// SIMATIC STEP 7 (V5.x) project Formation_tolerie
// CPU: CPU
// station: Matériel
// station: API
// station: P_ADR_BUS
// station: P_ADR_BUS
// station: Configuration
// station: MOP
// program: Programme S7(1)
// program: Programme S7(2)

SYMBOL_TABLE
"I01"	DB 1	FB 1	// FACILITY: INSTANCE DB (FB1)
"I02"	DB 2	FB 2	// FACILITY: INSTANCE DB FOR MMC CONTROL (FB2)
"I03"	DB 3	FB 3	// FACILITY: INSTANCE DB FOR MOP/LOP
"I04"	DB 4	FB 4	// FACILITY: INSTANCE DB FOR COMMUNICATION / DB D'INSTANCE POUR LA COMMUNICATION
"SFM_DB"	DB 75	FB 20	// Bloc de diagnostic pour signalisation d'erreurs système
"SFM_GLOBAL_DB"	DB 76	DB 76	// Bloc de diagnostic pour signalisation d'erreurs système
"SFM_PN"	DB 77	DB 77	// PROFINET DIAGNOSTIC FUNCTION EDITING DB FOR IHMP
"IDENT"	DB 93	DB 93	// RFID DATAS / IDENTIFIANT DYNAMIQUE
"IIT"	DB 96	DB 96	// FACILITY: PART TABLE / DB TABLE PIECE
"IIS"	DB 97	DB 97	// FACILITY: SUPPORT WORD TABLE / DB MOTS SUPPORT
"IG"	DB 99	DB 99	// FACILITY: GLOBAL DB / DB GLOBAL
"Z1"	DB 100	FB 100	// ZONE 1: INSTANCE DB
"Z1A0"	DB 101	FB 101	// A0 ROBOT INSTANCE DATA BLOC / BLOC DE DONNEES INSTANCE A0 ROBOT
"Z1A01"	DB 102	FB 102	// A01 PREHENSEUR INSTANCE DATA BLOC / BLOC DE DONNEES INSTANCE A01 PREHENSEUR
"Z1B0"	DB 103	FB 103	// B0 MONTAGE INSTANCE DATA BLOC / BLOC DE DONNEES INSTANCE B0 MONTAGE
"Z1C0C"	DB 104	FB 104	// C0C CHGT_MEUBLE INSTANCE DATA BLOC / BLOC DE DONNEES INSTANCE C0C CHGT_MEUBLE
"Z1H0D"	DB 105	FB 105	// H0D DCHGT_MEUBL INSTANCE DATA BLOC / BLOC DE DONNEES INSTANCE H0D DCHGT_MEUBL
"Z1T"	DB 198	DB 198	// ZONE 1: REFERENCE TIME FOR MOVEMENTS
"Z1G"	DB 199	DB 199	// ZONE 1: GLOBAL DB
"ITS0"	DB 1100	FB 1100	// ILOT : DB INSTANCE FB1100
"ITSZ1_AU_ES_FZ"	DB 1110	FB 1110	// Z1 : DB D'INSTANCE DU FB 1110
"ITSZ1VAR"	DB 1113	FB 1113	// Z1 : DB D'INSTANCE DU FB 1113
"TSM"	DB 1279	DB 1279	// STD - DB global pour la Tâche de Sécurité
"TSE_AMONT"	DB 1286	FB 1692	// STD - INSTANCE DB OF FB 1692 (F_SENDDP) SAFETY DATA SEND
"TSR_AMONT"	DB 1287	FB 1693	// STD - INSTANCE DB OF FB 1693 (F_RCVDP) SAFETY DATA RECEIVE
"TSE_AVAL"	DB 1288	FB 1692	// STD - INSTANCE DB OF FB 1692 (F_SENDDP) SAFETY DATA SEND
"TSR_AVAL"	DB 1289	FB 1693	// STD - INSTANCE DB OF FB 1693 (F_RCVDP) SAFETY DATA RECEIVE
"F_GLOBDB"	DB 1300	DB 1300
"F00471__Z1RB1_M05"	DB 1301	FB 1300
"F00477__Z1RB1_M06"	DB 1302	FB 1300
"F00203__Z1ZB_M07"	DB 1303	FB 1300
"F00209__Z1ZB_M08"	DB 1304	FB 1300
"F00215__Z1ZB_M09"	DB 1305	FB 1300
"F00303__Z1SPA1"	DB 1306	FB 1300
"AFF"	DB 1863	DB 1863	// SIEBERT DISPLAY STRING STORAGE / STOCKAGE MESSAGE AFFICHEUR SIEBERT
"DB_IHM_WINCC"	DB 1962	FB 1962	// FACILITY: HMI INTERFACING WINCCFLEXIBLE RT
"DB_MMC"	DB 2000	DB 2000	// BACKUP COPY AND RESTORE OF EXTERN MEMORY MAP (MMC)
"DB_PN"	DB 2036	FB 2036	// INSTANCE IO PROFINET DB
"0_01_ILOT"	FB 1	FB 1	// FACILITY: FACILITY MANAGEMENT
"0_02_MMC"	FB 2	FB 2	// FACILITY: BACKUP MANAGEMENT AND DATA RESTITUTION ON EXTERNAL MMC CARD
"0_03_XOP"	FB 3	FB 3	// FACILITY: MOP/LOP MANAGEMENT
"0_04_COM"	FB 4	FB 4	// FACILITY: COM CONTROL WITH SIPTOL / GESTION DE LA COMMUNICATION AVEC SIPTOL
"SFM_FB"	FB 20	FB 20	// Bloc de diagnostic pour signalisation d'erreurs système
"1_00_ZONE1"	FB 100	FB 100	// ZONE 1: ZONE CONTROL
"1_A0_ROBOT"	FB 101	FB 101	// A0 ROBOT FUNCTION BLOC / SECTION PROGRAMME A0 ROBOT
"1_A01_PREHENSEUR"	FB 102	FB 102	// A01 PREHENSEUR FUNCTION BLOC / SECTION PROGRAMME A01 PREHENSEUR
"1_B0_MONTAGE"	FB 103	FB 103	// B0 MONTAGE FUNCTION BLOC / SECTION PROGRAMME B0 MONTAGE
"1_C0C_CHGT_MEUBLE"	FB 104	FB 104	// C0C CHGT_MEUBLE FUNCTION BLOC / SECTION PROGRAMME C0C CHGT_MEUBLE
"1_H0D_DCHGT_MEUBL"	FB 105	FB 105	// H0D DCHGT_MEUBL FUNCTION BLOC / SECTION PROGRAMME H0D DCHGT_MEUBL
"F_TON"	FB 185	FB 185	// F_: Timer Switch On Delay
"F_TOF"	FB 186	FB 186	// F_: Timer Switch Off Delay
"TS0"	FB 1100	FB 1100	// ILOT: FB Gestion SAFETY ilot
"TSZ1_AU_ES_FZ"	FB 1110	FB 1110
"F_IO_CGP"	FB 1300	FB 1300
"F_CTRL_1"	FB 1301	FB 1301
"F_CTRL_2"	FB 1302	FB 1302
"FITON"	FB 1303	FB 1303
"FIACK_GL"	FB 1304	FB 1304
"F_DIAG_N"	FB 1306	FB 1306
"F_RTGCO2"	FB 1308	FB 1308
"BF_DEVERM"	FB 1649	FB 1649	// BF STAGE DRY RUN CONTROL / BF GESTION DEVERMINAGE POSTE
"BF_RB_NISSAN"	FB 1650	FB 1650	// FANUC NISSAN ROBOT FB / BF ROBOT FANUC NISSAN
"TUSEND"	FB 1681	FB 1681	// Send Data via UDP
"TCON"	FB 1685	FB 1685	// Connect
"F_SENDDP"	FB 1692	FB 1692	// F_: Send Data via PROFIBUS DP / PROFINET IO
"F_RCVDP"	FB 1693	FB 1693	// F_: Receive Data via PROFIBUS DP / PROFINET IO
"F_ACK_GL"	FB 1695	FB 1695	// Acquittement global de toutes les périphéries F d'un groupe d'exécution F
"P_SEND"	FB 1698	FB 1698	// Send Data to CP340
"P_RCV"	FB 1699	FB 1699	// Receive Data from CP340
"BFS_BSEC1"	FB 1710	FB 1710
"BFS_BSECTR1"	FB 1711	FB 1711
"BFS_PORTE1"	FB 1712	FB 1712
"BFS_AIR1"	FB 1713	FB 1713
"BFS_CRM1"	FB 1714	FB 1714
"BFS_CR1"	FB 1715	FB 1715
"BFS_CAME_ROBOT1"	FB 1716	FB 1716
"BFS_MUT1"	FB 1717	FB 1717
"BFS_BIMA"	FB 1719	FB 1719
"BFS_ROB_KUKA_PS"	FB 1720	FB 1720
"BF_PNPN_MESG"	FB 1852	FB 1852	// SEND RECEIVE MESSAGE BY PNPN INTERFACE/ EMISSION RECEPTION MESSAGE VIA PNPN
"BF_G120DS_V2"	FB 1853	FB 1853	// G120D DRIVE BOX CONTROL / GESTION COFFRET VAR G120D
"BF_G120S_V2"	FB 1854	FB 1854	// G120 DRIVE PLATE CONTROL / GESTION PLATINE VAR G120
"BF_CARACT_SIEBERT"	FB 1856	FB 1856	// SIEBERT DISPLAY MESSAGE CONFIGURATION / MISE EN FORME MESSAGE AFFICHEUR SIEBERT
"BF_AFF SIEBERT (2*13) PN"	FB 1860	FB 1860	// AFFICHEUR 2 LIGNES DE 13 CARACTERES
"BF_WELDING_BOX"	FB 1868	FB 1868	// WELDING BOX CONTROL / GESTION DES COFFRETS PARAMETRES SOUDURE
"BF_CONF_MACHINE"	FB 1869	FB 1869	// GESTION BASE DE DONNEE CONFIGURATION MACHINE
"BF_CODE_PROCESS"	FB 1870	FB 1870	// GESTION BASE DE DONNEE CODE PROCESS
"BF_DATABASE3"	FB 1871	FB 1871	// DATABASE MANAGEMENT / GESTION BASE DE DONNEES
"BF_IHMMUT1"	FB 1874	FB 1874	// Diagnostic IHM(P) BFS_MUT1
"BF_IHMCAME_ROBOT1"	FB 1875	FB 1875	// BF gérant le bon fonctionnement de la came robot
"BF_IHMCR1"	FB 1876	FB 1876	// BF gérant l'IHM du relais non piloté par l'API mais controlé
"BF_IHMCRM1"	FB 1877	FB 1877	// BF gérant l'IHM du relais de controçle raccordement de masse CRM
"BF_CABRS"	FB 1897	FB 1897	// BARCODE READER / LECTEUR DE CODE A BARRE
"BF_IHMPORTE1"	FB 1930	FB 1930	// BF - ZONE : Diagnostic du bloc BFS_IHMPORTE
"BF_IHMAIR1"	FB 1931	FB 1931	// BF - ZONE : Diagnostic du bloc BFS_IHMAIR
"BF_ZONE_MODE_IHM1"	FB 1932	FB 1932	// Zone: Traitement des Modes et des pupitre de cde manu de la  zone
"BF_RB_COD_PREH_API"	FB 1953	FB 1953	// Gestion du préhenseur par API (séquences 1 à 16)
"BF_MODBUS_MASTER_CP340"	FB 1958	FB 1958	// MODBUS MAITRE SUR CP 340 (LIAISON SERIE)
"BF_MODBUS_SLAVE_CP340"	FB 1959	FB 1959	// MODBUS ESCLAVE AVEC CP340
"BF_MODBUS_TCPIP_MASTER"	FB 1960	FB 1960	// BF gerant le protocole MODBUS TCP/IP en tant que Client TCP et Maitre MODBUS
"BF_MODBUS_TCPIP_SLAVE"	FB 1961	FB 1961	// ESCLAVE MODBUS SUR CP ETHERNET
"BF_IHM_WINCC"	FB 1962	FB 1962	// BF- GESTION IMAGES WINCC FLEXIBLE
"BF_RB_SERVICE"	FB 1997	FB 1997	// BF- Envoi d'un groupe de robot en rodage
"BF_MMC"	FB 2000	FB 2000	// SAUVEGARDE ET RESTITUTION MEMOIRE SUR CARTE MEMOIRE EXTERNE (MMC)
"BF_MB_CHAINE1"	FB 2001	FB 2001	// PILOTAGE DU MOTEUR DU MEUBLE ET SURVEILLANCE DES DEFAUTS
"BF_MB_BUTEE1"	FB 2002	FB 2002	// MEUBLE A ACCUMULATION - PILOTAGE D'UNE BUTEE
"BF_ILOT"	FB 2004	FB 2004	// BF- GESTION INFO LIE A L'INSTALLATION (ILOT)
"BF_B_VIEAPI"	FB 2006	FB 2006	// CONTRÔLE DE LA COMMUNICATION ENTRE DEUX AUTOMATES EN LIAISON
"BF_BUTEE_CONVOYEUR2"	FB 2007	FB 2007	// PILOTAGE D'UNE BUTEE
"BF_IDENT"	FB 2015	FB 2015	// LECTURE/ECRITURE DES ETIQUETTES RFID
"BF_ROBOT"	FB 2016	FB 2016	// Interface API - Robot Version 1.2a
"BF_TCY_SUIV"	FB 2019	FB 2019	// MESURE LES TEMPS DE CYCLE D'UN MOYEN DE PRODUCTION
"BF_RUP_FLU"	FB 2020	FB 2020	// SUIVI-RUPTURE DE FLUX
"BF_CPT_PIECE"	FB 2021	FB 2021	// BF- COMPTEUR DE PIECE
"BF_ACT_DESACT"	FB 2033	FB 2033	// BF- ACTIVATION DESACTIVATION D'UN IO DEVICE
"BF_DIAG_PROFINET"	FB 2036	FB 2036	// BF- DIAGNOSTIC PROFINET IO
"BF_TF_TP"	FB 2037	FB 2037	// TRANSFERT DE TABLE DE MEMOIRES PIECES
"BF_FIFO"	FB 2039	FB 2039	// ASSURE LA GESTION D'UNE PILE FIFO
"BF_MVSE2P1"	FB 2040	FB 2040	// GESTION D'UN MOUVEMENT SIMPLE EFFET 2 POSITIONS
"BF_MOUVMP1"	FB 2041	FB 2041	// GESTION D'UN MOUVEMENT MULTI POSITION
"BF_MOUV2P1"	FB 2042	FB 2042	// BF- GESTION D'UN MOUVEMENT A 2 POSITIONS
"0_00_CYCLE_ILOT"	FC 1	FC 1	// FACILITY: CALL OF FACILITY FB
"SFM_FC"	FC 22	FC 22	// Bloc de diagnostic pour signalisation d'erreurs système
"1_00_CYCLE_Z1"	FC 100	FC 100	// ZONE 1: CALL OF FB ZONE
"0_00_TSSAFETY"	FC 1100	FC 1100	// STD - FACILITY: EXECUTION F GROUP ASSOCIATE TO OB32 (NORMAL TASK)
"0_00_TSCYCLE"	FC 1101	FC 1101	// CALL OPERATOR NOT IN ZONE FB LINKED IN FACILITY
"C_CNTRL"	FC 1697	FC 1697	// Read Connection Diagnostic Information
"AG_SEND"	FC 1698	FC 1698	// AG SEND
"AG_RECV"	FC 1699	FC 1699	// AG RECEIVE
"BADI"	I 0.0	BOOL	// (MOP-IM.M01-02): BOUTON ANNULATION DEFAUT
"BRI"	I 0.1	BOOL	// (MOP-IM.M01-02): BOUTON REARMEMENT ILOT
"BMCY"	I 0.2	BOOL	// (MOP-IM.M01-02): BOUTON MARCHE CYCLE
"SMM"	I 0.3	BOOL	// (MOP-IM.M01-02): SELECTEUR MODE MANUEL
"SMA"	I 0.4	BOOL	// (MOP-IM.M01-02): SELECTEUR MODE AUTO
"Z1BMR1"	I 0.5	BOOL	// (MOP-IM.M01-02): BOUTON RECUL MOUVEMENT
"Z1BMA1"	I 0.6	BOOL	// (MOP-IM.M01-02): BOUTON AVANCE MOUVEMENT
"B0DAPL1"	I 78.0	BOOL	// (B0IM.B0E1): B0 DETECTEUR AVANCE PILOTE 1
"B0DAPL2"	I 78.1	BOOL	// (B0IM.B0E1): B0 DETECTEUR AVANCE PILOTE 2
"B0DFSR3"	I 78.2	BOOL	// (B0IM.B0E1): B0 DETECTEUR FERMETURE SERRAGE 3
"B0DFSR4"	I 78.3	BOOL	// (B0IM.B0E1): B0 DETECTION FERMETURE SERRAGE 4
"B0DRPL1"	I 78.4	BOOL	// (B0IM.B0E1): B0 DETECTEUR RECUL PILOTE 1
"B0DRPL2"	I 78.5	BOOL	// (B0IM.B0E1): B0 DETECTEUR RECUL PILOTE 2
"B0DOSR3"	I 78.6	BOOL	// (B0IM.B0E1): B0 DETECTEUR OUVERTURE SERRAGE 3
"B0DOSR4"	I 78.7	BOOL	// (B0IM.B0E1): B0 DETECTION OUVERTURE SERRAGE 4
"B0DPP"	I 79.0	BOOL	// (B0IM.B0E1): B0 DETECTEUR PRESENCE PIECE
"A01DFSR1"	I 80.0	BOOL	// (A01IM.E1): A01 DETECTEUR FERMETURE SERRAGE 1
"A01DFSR2"	I 80.1	BOOL	// (A01IM.E1): A01 DETECTEUR FERMETURE SERRAGE 2
"A01DFSR3"	I 80.2	BOOL	// (A01IM.E1): A01 DETECTEUR FERMETURE SERRAGE 3
"A01DOSR1"	I 80.4	BOOL	// (A01IM.E1): A01 DETECTEUR OUVERTURE SERRAGE 1
"A01DOSR2"	I 80.5	BOOL	// (A01IM.E1): A01 DETECTEUR OUVERTURE SERRAGE 2
"A01DOSR3"	I 80.6	BOOL	// (A01IM.E1): A01 DETECTEUR OUVERTURE SERRAGE 3
"A01DPP"	I 81.0	BOOL	// (A01IM.E1): A01 DETECTION PRESENCE PIECE
"Z1CCSC1"	I 200.0	BOOL	// (Z1ZB.M02): CONTROLE RETOUR COMMUN SECURITE AU (SC1)
"Z1CCES"	I 200.1	BOOL	// (Z1ZB.M02): CONTROLE RETOUR COMMUN SECURITE ES
"Z1CCFZ"	I 200.2	BOOL	// (Z1ZB.M02): CONTROLE RETOUR COMMUN SECURITE FZ
"Z1CCB24Z"	I 200.4	BOOL	// (Z1ZB.M02): RETOUR CONTROLE DISJONCTEUR 24V (24Z)
"Z1CCB24R"	I 200.5	BOOL	// (Z1ZB.M02): RETOUR CONTROLE DISJONCTEUR 24V (24R)
"Z1CCB24SC"	I 200.6	BOOL	// (Z1ZB.M02): RETOUR CONTROLE DISJONCTEUR 24V (SC)
"Z1CP7B"	I 201.0	BOOL	// (Z1ZB.M03): CONTROLE PRESSION 7 BARS
"Z1CRM"	I 201.1	BOOL	// (Z1ZB.M03): RETOUR RELAIS CONTROLE DE MASSE
"Z1BMCY"	I 202.0	BOOL	// (Z1ZB.M04): BOUTON MARCHE CYCLE
"BAUI"	I 203.0	BOOL	// (Z1ZB.M07): ARRET D'URGENCE ILOT
"Z1SSZ"	I 203.2	BOOL	// (Z1ZB.M07): SELECTEUR SECURITE ZONE
"Z1SPA1BMCY"	I 300.7	BOOL	// (Z1SPA1.I0): BOUTON MARCHE CYCLE
"Z1SPA1BDACY"	I 301.0	BOOL	// (Z1SPA1.I1): BOUTON DEMANDE ARRET CYCLE
"Z1SPA1SPES"	I 301.3	BOOL	// (Z1SPA1.I1): SELECTEUR EN SERVICE / HORS SERVICE PORTILLON
"Z1SPA1SS"	I 303.7	BOOL	// (Z1SPA1.SI0): SELECTEUR DE SECURITE
"Z1SPA1CFP"	I 304.0	BOOL	// (Z1SPA1.SI1): CONTROLE FERMETURE PORTE
"A0RC_READY"	I 350.0	BOOL	// (A0RB.E1): ROBOT PRET
"A0MOTORON"	I 350.1	BOOL	// (A0RB.E1): SOUS PUISSANCE
"A0AUTO"	I 350.2	BOOL	// (A0RB.E1): COMMUTATEUR EN AUTOMATIQUE
"A0MANU"	I 350.3	BOOL	// (A0RB.E1): COMMUTATEUR EN MANUEL
"A0REPLI"	I 350.4	BOOL	// (A0RB.E1): POSITION DE REPLI
"A0RAMVT"	I 350.7	BOOL	// (A0RB.E1): MOUVEMENT EN COURS
"A0HPR"	I 351.0	BOOL	// (A0RB.E1): HORS PRODUCTION
"A0AOP"	I 351.1	BOOL	// (A0RB.E1): APPEL OPERATEUR
"A0DE"	I 351.2	BOOL	// (A0RB.E1): DERIVE
"A0TC"	I 351.3	BOOL	// (A0RB.E1): TOP CYCLE
"A0AI"	I 351.4	BOOL	// (A0RB.E1): ARRET INDUIT
"A0APE"	I 351.5	BOOL	// (A0RB.E1): ARRET PROPRE EXPLOITATION
"A0APF"	I 351.6	BOOL	// (A0RB.E1): ARRET PROPRE FABRICATION
"A0APP"	I 351.7	BOOL	// (A0RB.E1): ARRET PROPRE PANNE
"A0OR1"	I 352.0	BOOL	// (A0RB.E2): ORDRE 1
"A0OR2"	I 352.1	BOOL	// (A0RB.E2): ORDRE 2
"A0OR3"	I 352.2	BOOL	// (A0RB.E2): ORDRE 3
"A0OR4"	I 352.3	BOOL	// (A0RB.E2): ORDRE 4
"A0OR5"	I 352.4	BOOL	// (A0RB.E2): ORDRE 5
"A0OR6"	I 352.5	BOOL	// (A0RB.E2): ORDRE 6
"A0OR7"	I 352.6	BOOL	// (A0RB.E2): ORDRE 7
"A0OR8"	I 352.7	BOOL	// (A0RB.E2): ORDRE 8
"A0OR9"	I 353.0	BOOL	// (A0RB.E2): ORDRE 9
"A0OR10"	I 353.1	BOOL	// (A0RB.E2): ORDRE 10
"A0OR11"	I 353.2	BOOL	// (A0RB.E2): ORDRE 11
"A0OR12"	I 353.3	BOOL	// (A0RB.E2): ORDRE 12
"A0OR13"	I 353.4	BOOL	// (A0RB.E2): ORDRE 13
"A0OR14"	I 353.5	BOOL	// (A0RB.E2): ORDRE 14
"A0OR15"	I 353.6	BOOL	// (A0RB.E2): ORDRE 15
"A0OR16"	I 353.7	BOOL	// (A0RB.E2): ORDRE 16
"A0CCHDE"	I 354.0	BOOL	// (A0RB.E3): INFO CHANGEUR DEVERROUILLE
"A0CCHVE"	I 354.1	BOOL	// (A0RB.E3): INFO CHANGEUR VERROUILLE
"A0CPO"	I 354.2	BOOL	// (A0RB.E3): DETECTEUR PRESENCE OUTIL
"A0CPADV"	I 354.3	BOOL	// (A0RB.E3): CONTROLE PRESSION D'AIR DE DEVERROUILLAGE
"A0CPAV"	I 354.4	BOOL	// (A0RB.E3): CONTROLE PRESSION D'AIR DE VERROUILLAGE
"A0CPAS"	I 354.5	BOOL	// (A0RB.E3): CONTROLE PRESSION D'AIR (EV DE SECURITE)
"A0COHSUP"	I 354.6	BOOL	// (A0RB.E3): CONTROLE OUTIL HORS SUPPORT
"A0CFRO_ES"	I 354.7	BOOL	// (A0RB.E3): CONTROLE FRO MISE EN SERVICE
"A0CFRO_ZF"	I 355.0	BOOL	// (A0RB.E3): CONTROLE FRO FERMETURE ZONE 1
"A0CPAIR"	I 355.1	BOOL	// (A0RB.E3): CONTROLE PRESSION AIR DU ROBOT
"A0P1KCP"	I 355.2	BOOL	// (A0RB.E3): KCP ROBOT - POIDS 1
"A0P2KCP"	I 355.3	BOOL	// (A0RB.E3): KCP ROBOT - POIDS 2
"A0P4KCP"	I 355.4	BOOL	// (A0RB.E3): KCP ROBOT - POIDS 4
"A0P8KCP"	I 355.5	BOOL	// (A0RB.E3): KCP ROBOT - POIDS 8
"A0P16KCP"	I 355.6	BOOL	// (A0RB.E3): KCP ROBOT - POIDS 16
"A0P32KCP"	I 355.7	BOOL	// (A0RB.E3): KCP ROBOT - POIDS 32
"A0ORO1"	I 358.0	BOOL	// (A0RB.E5): ORDRE OUTIL 1
"A0ORO2"	I 358.1	BOOL	// (A0RB.E5): ORDRE OUTIL 2
"A0ORO3"	I 358.2	BOOL	// (A0RB.E5): ORDRE OUTIL 3
"A0ORO4"	I 358.3	BOOL	// (A0RB.E5): ORDRE OUTIL 4
"A0ORO5"	I 358.4	BOOL	// (A0RB.E5): ORDRE OUTIL 5
"A0ORO6"	I 358.5	BOOL	// (A0RB.E5): ORDRE OUTIL 6
"A0ORO7"	I 358.6	BOOL	// (A0RB.E5): ORDRE OUTIL 7
"A0ORO8"	I 358.7	BOOL	// (A0RB.E5): ORDRE OUTIL 8
"A0ORO9"	I 359.0	BOOL	// (A0RB.E5): ORDRE OUTIL 9
"A0ORO10"	I 359.1	BOOL	// (A0RB.E5): ORDRE OUTIL 10
"A0ORO11"	I 359.2	BOOL	// (A0RB.E5): ORDRE OUTIL 11
"A0ORO12"	I 359.3	BOOL	// (A0RB.E5): ORDRE OUTIL 12
"A0ORO13"	I 359.4	BOOL	// (A0RB.E5): ORDRE OUTIL 13
"A0ORO14"	I 359.5	BOOL	// (A0RB.E5): ORDRE OUTIL 14
"A0ORO15"	I 359.6	BOOL	// (A0RB.E5): ORDRE OUTIL 15
"A0ORO16"	I 359.7	BOOL	// (A0RB.E5): ORDRE OUTIL 16
"A0OR17"	I 364.0	BOOL	// (A0RB.E8): ORDRE 17
"A0OR18"	I 364.1	BOOL	// (A0RB.E8): ORDRE 18
"A0OR19"	I 364.2	BOOL	// (A0RB.E8): ORDRE 19
"A0OR20"	I 364.3	BOOL	// (A0RB.E8): ORDRE 20
"A0OR21"	I 364.4	BOOL	// (A0RB.E8): ORDRE 21
"A0OR22"	I 364.5	BOOL	// (A0RB.E8): ORDRE 22
"A0OR23"	I 364.6	BOOL	// (A0RB.E8): ORDRE 23
"A0OR24"	I 364.7	BOOL	// (A0RB.E8): ORDRE 24
"A0OR25"	I 365.0	BOOL	// (A0RB.E8): ORDRE 25
"A0OR26"	I 365.1	BOOL	// (A0RB.E8): ORDRE 26
"A0OR27"	I 365.2	BOOL	// (A0RB.E8): ORDRE 27
"A0OR28"	I 365.3	BOOL	// (A0RB.E8): ORDRE 28
"A0OR29"	I 365.4	BOOL	// (A0RB.E8): ORDRE 29
"A0OR30"	I 365.5	BOOL	// (A0RB.E8): ORDRE 30
"A0OR31"	I 365.6	BOOL	// (A0RB.E8): ORDRE 31
"A0OR32"	I 365.7	BOOL	// (A0RB.E8): ORDRE 32
"C0CDOB1"	I 430.0	BOOL	// (C0CIM.E1): DETECTEUR OUVERTURE BUTEE 1
"C0CDSPB1"	I 430.1	BOOL	// (C0CIM.E1): DETECTEUR SUPPORT PRESENT BUTEE 1
"C0CDOB2"	I 430.2	BOOL	// (C0CIM.E1): DETECTEUR OUVERTURE BUTEE 2
"C0CDSPB2"	I 430.3	BOOL	// (C0CIM.E1): DETECTEUR SUPPORT PRESENT BUTEE 2
"C0CDFB1"	I 430.4	BOOL	// (C0CIM.E1): DETECTEUR FERMETURE BUTEE 1
"C0CDSMAX"	I 430.5	BOOL	// (C0CIM.E1): DETECTEUR SEUIL MAX
"C0CDFB2"	I 430.6	BOOL	// (C0CIM.E1): DETECTEUR FERMETURE BUTEE 2
"C0CDDZB2"	I 430.7	BOOL	// (C0CIM.E1): DETECTEUR DEVERROUILLAGE DE ZONE BUTEE 2
"C0DPP1B2"	I 431.0	BOOL	// (C0CIM.E2): DETECTEUR PRESENCE PIECE TYPE 1
"C0CSSC"	I 431.2	BOOL	// (C0CIM.E2): C0C SELECTEUR DE SECURITE
"C0DPP2B2"	I 431.4	BOOL	// (C0CIM.E2): DETECTEUR PRESENCE PIECE TYPE 2
"H0DSSD"	I 450.0	BOOL	// (H0DIM.I1): SELECTEUR DE SECURITE
"H0DDM1_OK"	I 451.0	BOOL	// (H0DIM.DME1): DEPART MOTEUR PRET
"H0DDM1_CDM"	I 451.1	BOOL	// (H0DIM.DME1): DEPART MOTEUR EN MARCHE
"H0DDM1_DF"	I 451.2	BOOL	// (H0DIM.DME1): DEPART MOTEUR EN DEFAUT
"H0DDM1_AL"	I 451.3	BOOL	// (H0DIM.DME1): DEPART MOTEUR EN ALARME
"H0DDOB8"	I 453.0	BOOL	// (H0DIM.E1): DETECTEUR OUVERTURE BUTEE 8
"H0DDSPB8"	I 453.1	BOOL	// (H0DIM.E1): DETECTEUR SUPPORT PRESENT BUTEE 8
"H0DDOB9"	I 453.2	BOOL	// (H0DIM.E1): DETECTEUR OUVERTURE BUTEE 9
"H0DDSPB9"	I 453.3	BOOL	// (H0DIM.E1): DETECTEUR SUPPORT PRESENT BUTEE 9
"H0DDFB8"	I 453.4	BOOL	// (H0DIM.E1): DETECTEUR FERMETURE BUTEE 8
"H0DDSIL"	I 453.5	BOOL	// (H0DIM.E1): DETECTEUR SILHOUETTE
"H0DDFB9"	I 453.6	BOOL	// (H0DIM.E1): DETECTEUR FERMETURE BUTEE 9
"H0DDDZB9"	I 453.7	BOOL	// (H0DIM.E1): DETECTEUR DEVERROUILLAGE DE ZONE BUTEE 9
"H0DPP1B9"	I 454.0	BOOL	// (H0DIM.E2): DETECTEUR PRESENCE PIECE TYPE 1
"H0DDSMIN"	I 454.2	BOOL	// (H0DIM.E2): DETECTEUR SEUIL MIN
"H0DSSP"	I 454.3	BOOL	// (H0DIM.E2): SELECTEUR DE SECURITE
"H0DPP2B9"	I 454.4	BOOL	// (H0DIM.E2): DETECTEUR PRESENCE PIECE TYPE 2
"H0DDSMAX"	I 454.6	BOOL	// (H0DIM.E2): DETECTEUR SEUIL MAX
"H0DLIMEF"	I 454.7	BOOL	// (H0DIM.E2): LIMITEUR D'EFFORT
"Z1RB1CCB24Z"	I 470.4	BOOL	// (Z1RB1.M02): RETOUR CONTROLE DISJONCTEUR 24V (24Z)
"Z1RB1CCB24R"	I 470.5	BOOL	// (Z1RB1.M02): RETOUR CONTROLE DISJONCTEUR 24V (24R)
"A0BAU"	I 471.0	BOOL	// (Z1RB1.M05): ARRET D'URGENCE ROBOT
"A0RBMS1"	IW 350	WORD	// WORD 1 GENERAL DATA / GENERALITES
"A0RBMS2"	IW 352	WORD	// WORD 2 ROBOT ORDERS / ORDRES ROBOT
"A0RBMS3"	IW 354	WORD	// WORD 3 GRIPPER AND TOOL CHANGER / PREHENSEUR ET CHANGEUR OUTIL
"A0RBMS4"	IW 356	WORD	// WORD 4 FAULT NUMBER / NUMERO DE DEFAUT
"A0RBMS5"	IW 358	WORD	// WORD 5 TOOL ORDERS/ ORDRES OUTIL
"A0RBMS6"	IW 360	WORD	// WORD 6
"A0RBMS7"	IW 362	WORD	// WORD 7
"A0RBMS8"	IW 364	WORD	// WORD 8
"BA0"	M 0.0	BOOL	// FACILITY: BIT ALWAYS OFF / ILOT: BIT TOUJOURS A 0
"BA1"	M 0.1	BOOL	// FACILITY: BIT ALWAYS ON / ILOT: BIT TOUJOURS A 1
"BA1LIEN"	M 0.2	BOOL	// FACILITY: BIT ALWAYS ON (LINK IN THE PROGRAMMING NETWORK)
"SHUNT"	M 0.3	BOOL	// BIT FOR BYPASS DURING FACILITY START UP / BIT SHUNT POUR LA MISE AU POINT
"PERSO"	M 0.4	BOOL	// NEED TO PERSONALIZE BY THE PROGRAMMER / EQUATION A PERSONNALISER
"POUB"	M 0.5	BOOL	// DUST BIN BIT / BIT POUBELLE
"SYSFROID"	M 0.7	BOOL	// DETECTING COLD START PLC (OB102) / DETECTION DEMARRAGE A FROID API (OB102)
"ICL080S"	M 1.4	BOOL	// BLINKING INFORMATION / INFORMATION CLIGNOTEMENT
"IADF"	M 10.1	BOOL	// FACILITY: FAULT RESET INFORMATION (SAFETY)
"IR"	M 10.2	BOOL	// FACILITY: CONTROL ON INFORMATION (SAFETY)
"Z1DEF_MAJ"	M 11.0	BOOL	// ZONE 1: MAJOR FAULT (SAFETY)
"Z1IADF"	M 11.1	BOOL	// ZONE 1: FAULT RESET INFORMATION (SAFETY)
"Z1IR"	M 11.2	BOOL	// ZONE 1: CONTROL ON INFORMATION (SAFETY)
"Z1IAFJ"	M 11.3	BOOL	// ZONE 1: END OF PRODUCTION STOP INFORMATION (SAFETY)
"Z1MAUTO"	M 11.4	BOOL	// ZONE 1: ZONE IN AUTOMATIC MODE (SAFETY)
"H0AV"	M 100.0	BOOL	// Pilotage chaine H0
"SIMU"	M 105.0	BOOL	// Mode simulation en cours
"CYCL_EXC"	OB 1	OB 1	// EXECUTION CYCLE
"CYC_INT4"	OB 34	OB 34	// CYCLIC INTERRUPT 4
"I/O_FLT1"	OB 82	OB 82	// I/O POINT FAULT 1
"I/O_FLT2"	OB 83	OB 83	// I/O POINT FAULT 2
"OBNL_FLT"	OB 85	OB 85	// OB NOT LOADED FAULT
"RACK_FLT"	OB 86	OB 86	// LOSS OF RACK FAULT
"COMPLETE RESTART"	OB 100	OB 100	// COMPLETE RESTART
"MOD_ERR"	OB 122	OB 122	// MODULE ACCESS ERROR
"VADI"	Q 0.0	BOOL	// (MOP-IM.M06-07): VOYANT ANNULATION DEFAUT
"VMCY"	Q 0.1	BOOL	// (MOP-IM.M06-07): VOYANT MARCHE CYCLE
"VAOP"	Q 0.3	BOOL	// (MOP-IM.M06-07): VERRINE APPEL OPERATEUR
"A01EFSR1"	Q 56.0	BOOL	// (A01IM.S1): EV FERMETURE SERRAGE 1
"A01EFSR2"	Q 56.1	BOOL	// (A01IM.S1): A01 EV FERMETURE SERRAGE 2
"A01EFSR3"	Q 56.2	BOOL	// (A01IM.S1): A01 EV FERMETURE SERRAGE 3
"A01EOSR1"	Q 56.4	BOOL	// (A01IM.S1): A01 OUVERTURE SERRAGE 1
"A01EOSR2"	Q 56.5	BOOL	// (A01IM.S1): A01 EV OUVERTURE SERRAGE 2
"A01EOSR3"	Q 56.6	BOOL	// (A01IM.S1): A01 EV OUVERTURE SERRAGE 3
"B0EAPL1"	Q 58.0	BOOL	// (B0IM.B0S1): B0 EV AVANCE PILOTE 1
"B0EAPL2"	Q 58.1	BOOL	// (B0IM.B0S1): B0 EV AVANCE PILOTE 2
"B0EFSR3"	Q 58.2	BOOL	// (B0IM.B0S1): B0 EV FERMETURE SERRAGE 3
"B0EFSR4"	Q 58.3	BOOL	// (B0IM.B0S1): B0 EV FERMETURE SERRAGE 4
"B0ERPL1"	Q 58.4	BOOL	// (B0IM.B0S1): B0 EV RECUL PILOTE 1
"B0ERPL2"	Q 58.5	BOOL	// (B0IM.B0S1): B0 EV RECUL PILOTE 2
"B0EOSR3"	Q 58.6	BOOL	// (B0IM.B0S1): B0 EV OUVERTURE SERRAGE 3
"B0EOSR4"	Q 58.7	BOOL	// (B0IM.B0S1): B0 EV OUVERTURE SERRAGE 4
"Z1VMCY"	Q 200.0	BOOL	// (Z1ZB.M05): VOYANT MARCHE CYCLE
"Z1RCM"	Q 200.7	BOOL	// (Z1ZB.M05): RELAIS DE CONTROLE DE MASSE
"Z1RSC1"	Q 215.0	BOOL	// (Z1ZB.M09): RELAI COMMUN DE SECURITE SC1
"Z1RES"	Q 215.1	BOOL	// (Z1ZB.M09): RELAI COMMUN DE SECURITE ES
"Z1RFZ"	Q 215.2	BOOL	// (Z1ZB.M09): RELAI COMMUN DE SECURITE FZ
"Z1SPA1VMCY"	Q 300.7	BOOL	// (Z1SPA1.O0): VOYANT MARCHE CYCLE
"Z1SPA1VDACY"	Q 301.0	BOOL	// (Z1SPA1.O1): VOYANT DEMANDE ARRET CYCLE
"A0AEVRB"	Q 350.0	BOOL	// (A0RB.S1): AUTORISATION D'EVOLUTION
"A0DMSP"	Q 350.1	BOOL	// (A0RB.S1): DEMANDE DE MISE SOUS PUISSANCE
"A0STOP"	Q 350.2	BOOL	// (A0RB.S1): ARRET ROBOT
"A0DDCY"	Q 350.3	BOOL	// (A0RB.S1): DEPART CYCLE
"A0DEV"	Q 350.4	BOOL	// (A0RB.S1): DEVERMINAGE
"A0CVC_0"	Q 350.5	BOOL	// (A0RB.S1): CONTROLE VALIDATION CODE A 0
"A0CVC_1"	Q 350.6	BOOL	// (A0RB.S1): CONTROLE VALIDATION CODE A 1
"A0CPCO"	Q 350.7	BOOL	// (A0RB.S1): CONTOLE PARITE CODE
"A0C1"	Q 351.0	BOOL	// (A0RB.S1): CODE POIDS 1
"A0C2"	Q 351.1	BOOL	// (A0RB.S1): CODE POIDS 2
"A0C4"	Q 351.2	BOOL	// (A0RB.S1): CODE POIDS 4
"A0C8"	Q 351.3	BOOL	// (A0RB.S1): CODE POIDS 8
"A0C16"	Q 351.4	BOOL	// (A0RB.S1): CODE POIDS 16
"A0C32"	Q 351.5	BOOL	// (A0RB.S1): CODE POIDS 32
"A0C64"	Q 351.6	BOOL	// (A0RB.S1): CODE POIDS 64
"A0C128"	Q 351.7	BOOL	// (A0RB.S1): CODE POIDS 128
"A0EV1"	Q 352.0	BOOL	// (A0RB.S2): EVENEMENT 1
"A0EV2"	Q 352.1	BOOL	// (A0RB.S2): EVENEMENT 2
"A0EV3"	Q 352.2	BOOL	// (A0RB.S2): EVENEMENT 3
"A0EV4"	Q 352.3	BOOL	// (A0RB.S2): EVENEMENT 4
"A0EV5"	Q 352.4	BOOL	// (A0RB.S2): EVENEMENT 5
"A0EV6"	Q 352.5	BOOL	// (A0RB.S2): EVENEMENT 6
"A0EV7"	Q 352.6	BOOL	// (A0RB.S2): EVENEMENT 7
"A0EV8"	Q 352.7	BOOL	// (A0RB.S2): EVENEMENT 8
"A0EV9"	Q 353.0	BOOL	// (A0RB.S2): EVENEMENT 9
"A0EV10"	Q 353.1	BOOL	// (A0RB.S2): EVENEMENT 10
"A0EV11"	Q 353.2	BOOL	// (A0RB.S2): EVENEMENT 11
"A0EV12"	Q 353.3	BOOL	// (A0RB.S2): EVENEMENT 12
"A0EV13"	Q 353.4	BOOL	// (A0RB.S2): EVENEMENT 13
"A0EV14"	Q 353.5	BOOL	// (A0RB.S2): EVENEMENT 14
"A0EV15"	Q 353.6	BOOL	// (A0RB.S2): EVENEMENT 15
"A0EV16"	Q 353.7	BOOL	// (A0RB.S2): EVENEMENT 16
"A0ENPRO"	Q 354.0	BOOL	// (A0RB.S3): EN PRODUCTION
"A0RFZ"	Q 354.1	BOOL	// (A0RB.S3): ZONE FERMEE
"A0GS1"	Q 356.0	BOOL	// (A0RB.S4): GROUPE SEQUENCE POIDS 1
"A0GS2"	Q 356.1	BOOL	// (A0RB.S4): GROUPE SEQUENCE POIDS 2
"A0GS4"	Q 356.2	BOOL	// (A0RB.S4): GROUPE SEQUENCE POIDS 4
"A0GS8"	Q 356.3	BOOL	// (A0RB.S4): GROUPE SEQUENCE POIDS 8
"A0E1_SRE"	Q 356.4	BOOL	// (A0RB.S4): INFO DETECTION RECUL SEQUENCE 1
"A0E1_SAV"	Q 356.5	BOOL	// (A0RB.S4): INFO DETECTION AVANCE SEQUENCE 1
"A0E2_SRE"	Q 356.6	BOOL	// (A0RB.S4): INFO DETECTION RECUL SEQUENCE 2
"A0E2_SAV"	Q 356.7	BOOL	// (A0RB.S4): INFO DETECTION AVANCE SEQUENCE 2
"A0DECH"	Q 357.0	BOOL	// (A0RB.S4): COMMANDE DEVERROUILLAGE CHANGEUR
"A0EVO1"	Q 358.0	BOOL	// (A0RB.S5): EVENEMENT OUTIL 1
"A0EVO2"	Q 358.1	BOOL	// (A0RB.S5): EVENEMENT OUTIL 2
"A0EVO3"	Q 358.2	BOOL	// (A0RB.S5): EVENEMENT OUTIL 3
"A0EVO4"	Q 358.3	BOOL	// (A0RB.S5): EVENEMENT OUTIL 4
"A0EVO5"	Q 358.4	BOOL	// (A0RB.S5): EVENEMENT OUTIL 5
"A0EVO6"	Q 358.5	BOOL	// (A0RB.S5): EVENEMENT OUTIL 6
"A0EVO7"	Q 358.6	BOOL	// (A0RB.S5): EVENEMENT OUTIL 7
"A0EVO8"	Q 358.7	BOOL	// (A0RB.S5): EVENEMENT OUTIL 8
"A0EVO9"	Q 359.0	BOOL	// (A0RB.S5): EVENEMENT OUTIL 9
"A0EVO10"	Q 359.1	BOOL	// (A0RB.S5): EVENEMENT OUTIL 10
"A0EVO11"	Q 359.2	BOOL	// (A0RB.S5): EVENEMENT OUTIL 11
"A0EVO12"	Q 359.3	BOOL	// (A0RB.S5): EVENEMENT OUTIL 12
"A0EVO13"	Q 359.4	BOOL	// (A0RB.S5): EVENEMENT OUTIL 13
"A0EVO14"	Q 359.5	BOOL	// (A0RB.S5): EVENEMENT OUTIL 14
"A0EVO15"	Q 359.6	BOOL	// (A0RB.S5): EVENEMENT OUTIL 15
"A0EVO16"	Q 359.7	BOOL	// (A0RB.S5): EVENEMENT OUTIL 16
"A0EV17"	Q 364.0	BOOL	// (A0RB.S8): EVENEMENT 17
"A0EV18"	Q 364.1	BOOL	// (A0RB.S8): EVENEMENT 18
"A0EV19"	Q 364.2	BOOL	// (A0RB.S8): EVENEMENT 19
"A0EV20"	Q 364.3	BOOL	// (A0RB.S8): EVENEMENT 20
"A0EV21"	Q 364.4	BOOL	// (A0RB.S8): EVENEMENT 21
"A0EV22"	Q 364.5	BOOL	// (A0RB.S8): EVENEMENT 22
"A0EV23"	Q 364.6	BOOL	// (A0RB.S8): EVENEMENT 23
"A0EV24"	Q 364.7	BOOL	// (A0RB.S8): EVENEMENT 24
"A0EV25"	Q 365.0	BOOL	// (A0RB.S8): EVENEMENT 25
"A0EV26"	Q 365.1	BOOL	// (A0RB.S8): EVENEMENT 26
"A0EV27"	Q 365.2	BOOL	// (A0RB.S8): EVENEMENT 27
"A0EV28"	Q 365.3	BOOL	// (A0RB.S8): EVENEMENT 28
"A0EV29"	Q 365.4	BOOL	// (A0RB.S8): EVENEMENT 29
"A0EV30"	Q 365.5	BOOL	// (A0RB.S8): EVENEMENT 30
"A0EV31"	Q 365.6	BOOL	// (A0RB.S8): EVENEMENT 31
"A0EV32"	Q 365.7	BOOL	// (A0RB.S8): EVENEMENT 32
"C0CEOB1"	Q 430.0	BOOL	// (C0CIM.S1): ELECTROVANNE OUVERTURE BUTEE 1
"C0CEOB2"	Q 430.1	BOOL	// (C0CIM.S1): ELECTROVANNE OUVERTURE BUTEE 2
"C0CEFB1"	Q 430.4	BOOL	// (C0CIM.S1): ELECTROVANNE FERMETURE BUTEE 1
"C0CEFB2"	Q 430.5	BOOL	// (C0CIM.S1): ELECTROVANNE FERMETURE BUTEE 2
"H0DDM1_OAV"	Q 451.0	BOOL	// (H0DIM.DMS1): RELAI MARCHE AVANCE DEPART MOTEUR
"H0DDM1_ORE"	Q 451.1	BOOL	// (H0DIM.DMS1): RELAI MARCHE RECUL DEPART MOTEUR
"H0DDM1_FRE"	Q 451.2	BOOL	// (H0DIM.DMS1): COMMANDE FREIN DEPART MOTEUR
"H0DDM1_IR"	Q 451.3	BOOL	// (H0DIM.DMS1): INFORMATION REARMEMENT DEPART MOTEUR
"H0DEOB8"	Q 453.0	BOOL	// (H0DIM.S1): ELECTROVANNE OUVERTURE BUTEE 8
"H0DEOB9"	Q 453.1	BOOL	// (H0DIM.S1): ELECTROVANNE OUVERTURE BUTEE 9
"H0DEFB8"	Q 453.4	BOOL	// (H0DIM.S1): ELECTROVANNE FERMETURE BUTEE 8
"H0DEFB9"	Q 453.5	BOOL	// (H0DIM.S1): ELECTROVANNE FERMETURE BUTEE 9
"A0RBME1"	QW 350	WORD	// WORD 1 GENERAL DATA AND CYCLE CODE / CODE CYCLE ET GENERALITES
"A0RBME2"	QW 352	WORD	// WORD 2 ROBOT EVENTS / EVENEMENTS ROBOT
"A0RBME3"	QW 354	WORD	// WORD 3 GENERAL DATAS / GENERALITES
"A0RBME4"	QW 356	WORD	// WORD 4 GRIPPER AND TOOL CHANGER / PREHENSEUR ET CHANGEUR OUTIL
"A0RBME5"	QW 358	WORD	// WORD 5 TOOL EVENTS / EVENEMENTS OUTIL
"A0RBME6"	QW 360	WORD	// WORD 6
"A0RBME7"	QW 362	WORD	// WORD 7
"A0RBME8"	QW 364	WORD	// WORD 8
"TP"	SFB 3	SFB 3	// GENERATE A PULSE
"TON"	SFB 4	SFB 4	// GENERATE AN ON DELAY
"TOF"	SFB 5	SFB 5	// GENERATE AN OFF DELAY
"RDREC"	SFB 52	SFB 52	// READ A PROCESS DATA RECORD
"WRREC"	SFB 53	SFB 53	// WRITE A PROCESS DATA RECORD
"RALRM"	SFB 54	SFB 54	// Receive Alarm Data
"SET_CLK"	SFC 0	SFC 0	// SET SYSTEM CLOCK
"READ_CLK"	SFC 1	SFC 1	// READ SYSTEM CLOCK
"RD_SINFO"	SFC 6	SFC 6	// READ OB START INFORMATION
"D_ACT_DP"	SFC 12	SFC 12	// DEACTIVATING AND ACTIVATING DP SLAVES
"DPRD_DAT"	SFC 14	SFC 14	// READ CONSISTENT DATA OF A STANDARD DP SLAVE
"DPWR_DAT"	SFC 15	SFC 15	// WRITE CONSISTENT DATA TO A STANDARD DP SLAVE
"ALARM_SQ"	SFC 17	SFC 17	// Generate Block-Related Messages with Acknowledgment
"BLKMOV"	SFC 20	SFC 20	// COPY VARIABLES
"FILL"	SFC 21	SFC 21	// INITIALIZE A MEMORY AREA
"TEST_DB"	SFC 24	SFC 24	// TEST DATA BLOCK
"DIS_AIRT"	SFC 41	SFC 41	// DELAY THE HIGHER PRIORITY INTERRUPTS AND ASYNCHRONOUS ERRORS
"EN_AIRT"	SFC 42	SFC 42	// ENABLE HIGHER PRIORITY INTERRUPTS AND ASYNCHRONOUS ERRORS
"STP"	SFC 46	SFC 46	// CHANGE THE CPU TO STOP
"RDSYSST"	SFC 51	SFC 51	// READ A SYSTEM STATUS LIST OR PARTIAL LIST
"WR_REC"	SFC 58	SFC 58	// WRITE DATA RECORD
"RD_REC"	SFC 59	SFC 59	// READ A DATA RECORD
"TIME_TCK"	SFC 64	SFC 64	// READ THE SYSTEM TIME
"GEO_LOG"	SFC 70	SFC 70	// DETERMINE LOGICAL ADDRESS
"READ_DBL"	SFC 83	SFC 83	// READ DATA BLOCK OUT OF LOAD MEMORY
"WRIT_DBL"	SFC 84	SFC 84	// WRITE DATA BLOCK IN LOAD MEMORY
"DEL_SI"	SFC 106	SFC 106	// Deleting Dynamically Assigned System Instances
"ALARM_DQ"	SFC 107	SFC 107	// Creating Acknowledgeable Block-related Message
"ALARM_D"	SFC 108	SFC 108	// Creating Acknowledged Block-related Message
"LIEN_PUP"	UDT 1988	UDT 1988	// Gestion des Modes et des pupitres de cde manu de la  zone (BF_ZONE_MODE_IHM)
"LIEN_ILOT"	UDT 2004	UDT 2004	// INFO CONTROL LINKED TO THE FACILITY (BF_ILOT)
"MOT_FONC_MP"	UDT 2041	UDT 2041	// INFO CONTROL OF A MOVEMENT (BF_MOUVMP1)
"MOT_FONC"	UDT 2042	UDT 2042	// INFO D'UN MOUVEMENT (BF_MOUV2P1,BF_MVSE2P1, BF_RB_COD_PREH_API)
"VAT_SIMU"	VAT 1	
"Essais"	VAT 2	
END_SYMBOL_TABLE

SYMBOL_TABLE
"I01"	DB 1	FB 1	// FACILITY: INSTANCE DB (FB1)
"I02"	DB 2	FB 2	// FACILITY: INSTANCE DB FOR MMC CONTROL (FB2)
"I03"	DB 3	FB 3	// FACILITY: INSTANCE DB FOR MOP/LOP
"I04"	DB 4	FB 4	// FACILITY: INSTANCE DB FOR COMMUNICATION / DB D'INSTANCE POUR LA COMMUNICATION
"SFM_DB"	DB 75	FB 20	// FACILITY: DB FAILURE MESSAGE (SFM_FB) LINK WITH PROFINET CONTROL
"SFM_GLOBAL_DB"	DB 76	DB 76	// DIAGNOSTIC BLOCK FOR THE SIGNALISATION OF THE SYSTEM ERRORS
"SFM_PN"	DB 77	DB 77	// PROFINET DIAGNOSTIC FUNCTION EDITING DB FOR IHMP
"IDENT"	DB 93	DB 93	// RFID DATAS / IDENTIFIANT DYNAMIQUE
"IIT"	DB 96	DB 96	// FACILITY: PART TABLE / DB TABLE PIECE
"IIS"	DB 97	DB 97	// FACILITY: SUPPORT WORD TABLE / DB MOTS SUPPORT
"IG"	DB 99	DB 99	// FACILITY: GLOBAL DB / DB GLOBAL
"Z1"	DB 100	FB 100	// ZONE 1: INSTANCE DB
"Z1A0"	DB 101	FB 101	// A0 ROBOT INSTANCE DATA BLOC / BLOC DE DONNEES INSTANCE A0 ROBOT
"Z1A01"	DB 102	FB 102	// A01 PREHENSEUR INSTANCE DATA BLOC / BLOC DE DONNEES INSTANCE A01 PREHENSEUR
"Z1B0"	DB 103	FB 103	// B0 MONTAGE INSTANCE DATA BLOC / BLOC DE DONNEES INSTANCE B0 MONTAGE
"Z1C0C"	DB 104	FB 104	// C0C CHGT_MEUBLE INSTANCE DATA BLOC / BLOC DE DONNEES INSTANCE C0C CHGT_MEUBLE
"Z1H0D"	DB 105	FB 105	// H0D DCHGT_MEUBL INSTANCE DATA BLOC / BLOC DE DONNEES INSTANCE H0D DCHGT_MEUBL
"Z1T"	DB 198	DB 198	// ZONE 1: REFERENCE TIME FOR MOVEMENTS
"Z1G"	DB 199	DB 199	// ZONE 1: GLOBAL DB
"ITS0"	DB 1100	FB 1100	// ILOT : DB INSTANCE FB1100
"ITSZ1_AU_ES_FZ"	DB 1110	FB 1110	// Z1 : DB D'INSTANCE DU FB 1110
"ITSZ1VAR"	DB 1113	FB 1113	// Z1 : DB D'INSTANCE DU FB 1113
"TSM"	DB 1279	DB 1279	// STD - DB global pour la Tâche de Sécurité
"TSE_AMONT"	DB 1286	FB 1692	// STD - INSTANCE DB OF FB 1692 (F_SENDDP) SAFETY DATA SEND
"TSR_AMONT"	DB 1287	FB 1693	// STD - INSTANCE DB OF FB 1693 (F_RCVDP) SAFETY DATA RECEIVE
"TSE_AVAL"	DB 1288	FB 1692	// STD - INSTANCE DB OF FB 1692 (F_SENDDP) SAFETY DATA SEND
"TSR_AVAL"	DB 1289	FB 1693	// STD - INSTANCE DB OF FB 1693 (F_RCVDP) SAFETY DATA RECEIVE
"F_GLOBDB"	DB 1300	DB 1300
"F00471__Z1RB1_M05"	DB 1301	FB 1300
"F00477__Z1RB1_M06"	DB 1302	FB 1300
"F00203__Z1ZB_M07"	DB 1303	FB 1300
"F00209__Z1ZB_M08"	DB 1304	FB 1300
"F00215__Z1ZB_M09"	DB 1305	FB 1300
"F00303__Z1SPA1"	DB 1306	FB 1300
"AFF"	DB 1863	DB 1863	// SIEBERT DISPLAY STRING STORAGE / STOCKAGE MESSAGE AFFICHEUR SIEBERT
"DB_IHM_WINCC"	DB 1962	FB 1962	// FACILITY: HMI INTERFACING WINCCFLEXIBLE RT
"DB_MMC"	DB 2000	DB 2000	// BACKUP COPY AND RESTORE OF EXTERN MEMORY MAP (MMC)
"DB_PN"	DB 2036	FB 2036	// INSTANCE IO PROFINET DB
"0_01_ILOT"	FB 1	FB 1	// FACILITY: FACILITY MANAGEMENT
"0_02_MMC"	FB 2	FB 2	// FACILITY: BACKUP MANAGEMENT AND DATA RESTITUTION ON EXTERNAL MMC CARD
"0_03_XOP"	FB 3	FB 3	// FACILITY: MOP/LOP MANAGEMENT
"0_04_COM"	FB 4	FB 4	// FACILITY: COM CONTROL WITH SIPTOL / GESTION DE LA COMMUNICATION AVEC SIPTOL
"SFM_FB"	FB 20	FB 20	// DIAGNOSTIC BLOCK FOR SYSTEM ERRORS SIGNALLING
"1_00_ZONE1"	FB 100	FB 100	// ZONE 1: ZONE CONTROL
"1_A0_ROBOT"	FB 101	FB 101	// A0 ROBOT FUNCTION BLOC / SECTION PROGRAMME A0 ROBOT
"1_A01_PREHENSEUR"	FB 102	FB 102	// A01 PREHENSEUR FUNCTION BLOC / SECTION PROGRAMME A01 PREHENSEUR
"1_B0_MONTAGE"	FB 103	FB 103	// B0 MONTAGE FUNCTION BLOC / SECTION PROGRAMME B0 MONTAGE
"1_C0C_CHGT_MEUBLE"	FB 104	FB 104	// C0C CHGT_MEUBLE FUNCTION BLOC / SECTION PROGRAMME C0C CHGT_MEUBLE
"1_H0D_DCHGT_MEUBL"	FB 105	FB 105	// H0D DCHGT_MEUBL FUNCTION BLOC / SECTION PROGRAMME H0D DCHGT_MEUBL
"F_TON"	FB 185	FB 185	// F_: Timer Switch On Delay
"F_TOF"	FB 186	FB 186	// F_: Timer Switch Off Delay
"TS0"	FB 1100	FB 1100	// ILOT: FB Gestion SAFETY ilot
"TSZ1_AU_ES_FZ"	FB 1110	FB 1110
"F_IO_CGP"	FB 1300	FB 1300
"F_CTRL_1"	FB 1301	FB 1301
"F_CTRL_2"	FB 1302	FB 1302
"FITON"	FB 1303	FB 1303
"FIACK_GL"	FB 1304	FB 1304
"F_DIAG_N"	FB 1306	FB 1306
"F_RTGCO2"	FB 1308	FB 1308
"BF_DEVERM"	FB 1649	FB 1649	// BF STAGE DRY RUN CONTROL / BF GESTION DEVERMINAGE POSTE
"BF_RB_NISSAN"	FB 1650	FB 1650	// FANUC NISSAN ROBOT FB / BF ROBOT FANUC NISSAN
"TUSEND"	FB 1681	FB 1681	// Send Data via UDP
"TCON"	FB 1685	FB 1685	// Connect
"F_SENDDP"	FB 1692	FB 1692	// F_: Send Data via PROFIBUS DP / PROFINET IO
"F_RCVDP"	FB 1693	FB 1693	// F_: Receive Data via PROFIBUS DP / PROFINET IO
"F_ACK_GL"	FB 1695	FB 1695	// Acquittement global de toutes les périphéries F d'un groupe d'exécution F
"P_SEND"	FB 1698	FB 1698	// Send Data to CP340
"P_RCV"	FB 1699	FB 1699	// Receive Data from CP340
"BFS_BSEC1"	FB 1710	FB 1710
"BFS_BSECTR1"	FB 1711	FB 1711
"BFS_PORTE1"	FB 1712	FB 1712
"BFS_AIR1"	FB 1713	FB 1713
"BFS_CRM1"	FB 1714	FB 1714
"BFS_CR1"	FB 1715	FB 1715
"BFS_CAME_ROBOT1"	FB 1716	FB 1716
"BFS_MUT1"	FB 1717	FB 1717
"BFS_BIMA"	FB 1719	FB 1719
"BFS_ROB_KUKA_PS"	FB 1720	FB 1720
"BF_PNPN_MESG"	FB 1852	FB 1852	// SEND RECEIVE MESSAGE BY PNPN INTERFACE/ EMISSION RECEPTION MESSAGE VIA PNPN
"BF_G120DS_V2"	FB 1853	FB 1853	// G120D DRIVE BOX CONTROL / GESTION COFFRET VAR G120D
"BF_G120S_V2"	FB 1854	FB 1854	// G120 DRIVE PLATE CONTROL / GESTION PLATINE VAR G120
"BF_CARACT_SIEBERT"	FB 1856	FB 1856	// SIEBERT DISPLAY MESSAGE CONFIGURATION / MISE EN FORME MESSAGE AFFICHEUR SIEBERT
"BF_AFF SIEBERT (2*13) PN"	FB 1860	FB 1860	// AFFICHEUR 2 LIGNES DE 13 CARACTERES
"BF_WELDING_BOX"	FB 1868	FB 1868	// WELDING BOX CONTROL / GESTION DES COFFRETS PARAMETRES SOUDURE
"BF_CONF_MACHINE"	FB 1869	FB 1869	// GESTION BASE DE DONNEE CONFIGURATION MACHINE
"BF_CODE_PROCESS"	FB 1870	FB 1870	// GESTION BASE DE DONNEE CODE PROCESS
"BF_DATABASE3"	FB 1871	FB 1871	// DATABASE MANAGEMENT / GESTION BASE DE DONNEES
"BF_IHMMUT1"	FB 1874	FB 1874	// Diagnostic IHM(P) BFS_MUT1
"BF_IHMCAME_ROBOT1"	FB 1875	FB 1875	// BF gérant le bon fonctionnement de la came robot
"BF_IHMCR1"	FB 1876	FB 1876	// BF gérant l'IHM du relais non piloté par l'API mais controlé
"BF_IHMCRM1"	FB 1877	FB 1877	// BF gérant l'IHM du relais de controçle raccordement de masse CRM
"BF_CABRS"	FB 1897	FB 1897	// BARCODE READER / LECTEUR DE CODE A BARRE
"BF_IHMPORTE1"	FB 1930	FB 1930	// BF - ZONE : Diagnostic du bloc BFS_IHMPORTE
"BF_IHMAIR1"	FB 1931	FB 1931	// BF - ZONE : Diagnostic du bloc BFS_IHMAIR
"BF_ZONE_MODE_IHM1"	FB 1932	FB 1932	// Zone: Traitement des Modes et des pupitre de cde manu de la  zone
"BF_RB_COD_PREH_API"	FB 1953	FB 1953	// Gestion du préhenseur par API (séquences 1 à 16)
"BF_MODBUS_MASTER_CP340"	FB 1958	FB 1958	// MODBUS MAITRE SUR CP 340 (LIAISON SERIE)
"BF_MODBUS_SLAVE_CP340"	FB 1959	FB 1959	// MODBUS ESCLAVE AVEC CP340
"BF_MODBUS_TCPIP_MASTER"	FB 1960	FB 1960	// BF gerant le protocole MODBUS TCP/IP en tant que Client TCP et Maitre MODBUS
"BF_MODBUS_TCPIP_SLAVE"	FB 1961	FB 1961	// ESCLAVE MODBUS SUR CP ETHERNET
"BF_IHM_WINCC"	FB 1962	FB 1962	// BF- GESTION IMAGES WINCC FLEXIBLE
"BF_RB_SERVICE"	FB 1997	FB 1997	// BF- Envoi d'un groupe de robot en rodage
"BF_MMC"	FB 2000	FB 2000	// SAUVEGARDE ET RESTITUTION MEMOIRE SUR CARTE MEMOIRE EXTERNE (MMC)
"BF_MB_CHAINE1"	FB 2001	FB 2001	// PILOTAGE DU MOTEUR DU MEUBLE ET SURVEILLANCE DES DEFAUTS
"BF_MB_BUTEE1"	FB 2002	FB 2002	// MEUBLE A ACCUMULATION - PILOTAGE D'UNE BUTEE
"BF_ILOT"	FB 2004	FB 2004	// BF- GESTION INFO LIE A L'INSTALLATION (ILOT)
"BF_B_VIEAPI"	FB 2006	FB 2006	// CONTRÔLE DE LA COMMUNICATION ENTRE DEUX AUTOMATES EN LIAISON
"BF_BUTEE_CONVOYEUR2"	FB 2007	FB 2007	// PILOTAGE D'UNE BUTEE
"BF_IDENT"	FB 2015	FB 2015	// LECTURE/ECRITURE DES ETIQUETTES RFID
"BF_ROBOT"	FB 2016	FB 2016	// Interface API - Robot Version 1.2a
"BF_TCY_SUIV"	FB 2019	FB 2019	// MESURE LES TEMPS DE CYCLE D'UN MOYEN DE PRODUCTION
"BF_RUP_FLU"	FB 2020	FB 2020	// SUIVI-RUPTURE DE FLUX
"BF_CPT_PIECE"	FB 2021	FB 2021	// BF- COMPTEUR DE PIECE
"BF_ACT_DESACT"	FB 2033	FB 2033	// BF- ACTIVATION DESACTIVATION D'UN IO DEVICE
"BF_DIAG_PROFINET"	FB 2036	FB 2036	// BF- DIAGNOSTIC PROFINET IO
"BF_TF_TP"	FB 2037	FB 2037	// TRANSFERT DE TABLE DE MEMOIRES PIECES
"BF_FIFO"	FB 2039	FB 2039	// ASSURE LA GESTION D'UNE PILE FIFO
"BF_MVSE2P1"	FB 2040	FB 2040	// GESTION D'UN MOUVEMENT SIMPLE EFFET 2 POSITIONS
"BF_MOUVMP1"	FB 2041	FB 2041	// GESTION D'UN MOUVEMENT MULTI POSITION
"BF_MOUV2P1"	FB 2042	FB 2042	// BF- GESTION D'UN MOUVEMENT A 2 POSITIONS
"0_00_CYCLE_ILOT"	FC 1	FC 1	// FACILITY: CALL OF FACILITY FB
"SFM_FC"	FC 22	FC 22	// BLOCK DIAGNOSTIC FOR ERROR REPORTING SYSTEM
"1_00_CYCLE_Z1"	FC 100	FC 100	// ZONE 1: CALL OF FB ZONE
"0_00_TSSAFETY"	FC 1100	FC 1100	// STD - FACILITY: EXECUTION F GROUP ASSOCIATE TO OB32 (NORMAL TASK)
"0_00_TSCYCLE"	FC 1101	FC 1101	// CALL OPERATOR NOT IN ZONE FB LINKED IN FACILITY
"C_CNTRL"	FC 1697	FC 1697	// Read Connection Diagnostic Information
"AG_SEND"	FC 1698	FC 1698	// AG SEND
"AG_RECV"	FC 1699	FC 1699	// AG RECEIVE
"BADI"	I 0.0	BOOL	// (MOP-IM.M01-02): BOUTON ANNULATION DEFAUT
"BRI"	I 0.1	BOOL	// (MOP-IM.M01-02): BOUTON REARMEMENT ILOT
"BMCY"	I 0.2	BOOL	// (MOP-IM.M01-02): BOUTON MARCHE CYCLE
"SMM"	I 0.3	BOOL	// (MOP-IM.M01-02): SELECTEUR MODE MANUEL
"SMA"	I 0.4	BOOL	// (MOP-IM.M01-02): SELECTEUR MODE AUTO
"Z1BMR1"	I 0.5	BOOL	// (MOP-IM.M01-02): BOUTON RECUL MOUVEMENT
"Z1BMA1"	I 0.6	BOOL	// (MOP-IM.M01-02): BOUTON AVANCE MOUVEMENT
"B0DAPL1"	I 78.0	BOOL	// (B0IM.B0E1): B0 DETECTEUR AVANCE PILOTE 1
"B0DAPL2"	I 78.1	BOOL	// (B0IM.B0E1): B0 DETECTEUR AVANCE PILOTE 2
"B0DFSR3"	I 78.2	BOOL	// (B0IM.B0E1): B0 DETECTEUR FERMETURE SERRAGE 3
"B0DFSR4"	I 78.3	BOOL	// (B0IM.B0E1): B0 DETECTION FERMETURE SERRAGE 4
"B0DRPL1"	I 78.4	BOOL	// (B0IM.B0E1): B0 DETECTEUR RECUL PILOTE 1
"B0DRPL2"	I 78.5	BOOL	// (B0IM.B0E1): B0 DETECTEUR RECUL PILOTE 2
"B0DOSR3"	I 78.6	BOOL	// (B0IM.B0E1): B0 DETECTEUR OUVERTURE SERRAGE 3
"B0DOSR4"	I 78.7	BOOL	// (B0IM.B0E1): B0 DETECTION OUVERTURE SERRAGE 4
"B0DPP"	I 79.0	BOOL	// (B0IM.B0E1): B0 DETECTEUR PRESENCE PIECE
"A01DFSR1"	I 80.0	BOOL	// (A01IM.E1): A01 DETECTEUR FERMETURE SERRAGE 1
"A01DFSR2"	I 80.1	BOOL	// (A01IM.E1): A01 DETECTEUR FERMETURE SERRAGE 2
"A01DFSR3"	I 80.2	BOOL	// (A01IM.E1): A01 DETECTEUR FERMETURE SERRAGE 3
"A01DOSR1"	I 80.4	BOOL	// (A01IM.E1): A01 DETECTEUR OUVERTURE SERRAGE 1
"A01DOSR2"	I 80.5	BOOL	// (A01IM.E1): A01 DETECTEUR OUVERTURE SERRAGE 2
"A01DOSR3"	I 80.6	BOOL	// (A01IM.E1): A01 DETECTEUR OUVERTURE SERRAGE 3
"A01DPP"	I 81.0	BOOL	// (A01IM.E1): A01 DETECTION PRESENCE PIECE
"Z1CCSC1"	I 200.0	BOOL	// (Z1ZB.M02): CONTROLE RETOUR COMMUN SECURITE AU (SC1)
"Z1CCES"	I 200.1	BOOL	// (Z1ZB.M02): CONTROLE RETOUR COMMUN SECURITE ES
"Z1CCFZ"	I 200.2	BOOL	// (Z1ZB.M02): CONTROLE RETOUR COMMUN SECURITE FZ
"Z1CCB24Z"	I 200.4	BOOL	// (Z1ZB.M02): RETOUR CONTROLE DISJONCTEUR 24V (24Z)
"Z1CCB24R"	I 200.5	BOOL	// (Z1ZB.M02): RETOUR CONTROLE DISJONCTEUR 24V (24R)
"Z1CCB24SC"	I 200.6	BOOL	// (Z1ZB.M02): RETOUR CONTROLE DISJONCTEUR 24V (SC)
"Z1CP7B"	I 201.0	BOOL	// (Z1ZB.M03): CONTROLE PRESSION 7 BARS
"Z1CRM"	I 201.1	BOOL	// (Z1ZB.M03): RETOUR RELAIS CONTROLE DE MASSE
"Z1BMCY"	I 202.0	BOOL	// (Z1ZB.M04): BOUTON MARCHE CYCLE
"BAUI"	I 203.0	BOOL	// (Z1ZB.M07): ARRET D'URGENCE ILOT
"Z1SSZ"	I 203.2	BOOL	// (Z1ZB.M07): SELECTEUR SECURITE ZONE
"Z1SPA1BMCY"	I 300.7	BOOL	// (Z1SPA1.I0): BOUTON MARCHE CYCLE
"Z1SPA1BDACY"	I 301.0	BOOL	// (Z1SPA1.I1): BOUTON DEMANDE ARRET CYCLE
"Z1SPA1SPES"	I 301.3	BOOL	// (Z1SPA1.I1): SELECTEUR EN SERVICE / HORS SERVICE PORTILLON
"Z1SPA1SS"	I 303.7	BOOL	// (Z1SPA1.SI0): SELECTEUR DE SECURITE
"Z1SPA1CFP"	I 304.0	BOOL	// (Z1SPA1.SI1): CONTROLE FERMETURE PORTE
"A0RC_READY"	I 350.0	BOOL	// (A0RB.E1): ROBOT PRET
"A0MOTORON"	I 350.1	BOOL	// (A0RB.E1): SOUS PUISSANCE
"A0AUTO"	I 350.2	BOOL	// (A0RB.E1): COMMUTATEUR EN AUTOMATIQUE
"A0MANU"	I 350.3	BOOL	// (A0RB.E1): COMMUTATEUR EN MANUEL
"A0REPLI"	I 350.4	BOOL	// (A0RB.E1): POSITION DE REPLI
"A0RAMVT"	I 350.7	BOOL	// (A0RB.E1): MOUVEMENT EN COURS
"A0HPR"	I 351.0	BOOL	// (A0RB.E1): HORS PRODUCTION
"A0AOP"	I 351.1	BOOL	// (A0RB.E1): APPEL OPERATEUR
"A0DE"	I 351.2	BOOL	// (A0RB.E1): DERIVE
"A0TC"	I 351.3	BOOL	// (A0RB.E1): TOP CYCLE
"A0AI"	I 351.4	BOOL	// (A0RB.E1): ARRET INDUIT
"A0APE"	I 351.5	BOOL	// (A0RB.E1): ARRET PROPRE EXPLOITATION
"A0APF"	I 351.6	BOOL	// (A0RB.E1): ARRET PROPRE FABRICATION
"A0APP"	I 351.7	BOOL	// (A0RB.E1): ARRET PROPRE PANNE
"A0OR1"	I 352.0	BOOL	// (A0RB.E2): ORDRE 1
"A0OR2"	I 352.1	BOOL	// (A0RB.E2): ORDRE 2
"A0OR3"	I 352.2	BOOL	// (A0RB.E2): ORDRE 3
"A0OR4"	I 352.3	BOOL	// (A0RB.E2): ORDRE 4
"A0OR5"	I 352.4	BOOL	// (A0RB.E2): ORDRE 5
"A0OR6"	I 352.5	BOOL	// (A0RB.E2): ORDRE 6
"A0OR7"	I 352.6	BOOL	// (A0RB.E2): ORDRE 7
"A0OR8"	I 352.7	BOOL	// (A0RB.E2): ORDRE 8
"A0OR9"	I 353.0	BOOL	// (A0RB.E2): ORDRE 9
"A0OR10"	I 353.1	BOOL	// (A0RB.E2): ORDRE 10
"A0OR11"	I 353.2	BOOL	// (A0RB.E2): ORDRE 11
"A0OR12"	I 353.3	BOOL	// (A0RB.E2): ORDRE 12
"A0OR13"	I 353.4	BOOL	// (A0RB.E2): ORDRE 13
"A0OR14"	I 353.5	BOOL	// (A0RB.E2): ORDRE 14
"A0OR15"	I 353.6	BOOL	// (A0RB.E2): ORDRE 15
"A0OR16"	I 353.7	BOOL	// (A0RB.E2): ORDRE 16
"A0CCHDE"	I 354.0	BOOL	// (A0RB.E3): INFO CHANGEUR DEVERROUILLE
"A0CCHVE"	I 354.1	BOOL	// (A0RB.E3): INFO CHANGEUR VERROUILLE
"A0CPO"	I 354.2	BOOL	// (A0RB.E3): DETECTEUR PRESENCE OUTIL
"A0CPADV"	I 354.3	BOOL	// (A0RB.E3): CONTROLE PRESSION D'AIR DE DEVERROUILLAGE
"A0CPAV"	I 354.4	BOOL	// (A0RB.E3): CONTROLE PRESSION D'AIR DE VERROUILLAGE
"A0CPAS"	I 354.5	BOOL	// (A0RB.E3): CONTROLE PRESSION D'AIR (EV DE SECURITE)
"A0COHSUP"	I 354.6	BOOL	// (A0RB.E3): CONTROLE OUTIL HORS SUPPORT
"A0CFRO_ES"	I 354.7	BOOL	// (A0RB.E3): CONTROLE FRO MISE EN SERVICE
"A0CFRO_ZF"	I 355.0	BOOL	// (A0RB.E3): CONTROLE FRO FERMETURE ZONE 1
"A0CPAIR"	I 355.1	BOOL	// (A0RB.E3): CONTROLE PRESSION AIR DU ROBOT
"A0P1KCP"	I 355.2	BOOL	// (A0RB.E3): KCP ROBOT - POIDS 1
"A0P2KCP"	I 355.3	BOOL	// (A0RB.E3): KCP ROBOT - POIDS 2
"A0P4KCP"	I 355.4	BOOL	// (A0RB.E3): KCP ROBOT - POIDS 4
"A0P8KCP"	I 355.5	BOOL	// (A0RB.E3): KCP ROBOT - POIDS 8
"A0P16KCP"	I 355.6	BOOL	// (A0RB.E3): KCP ROBOT - POIDS 16
"A0P32KCP"	I 355.7	BOOL	// (A0RB.E3): KCP ROBOT - POIDS 32
"A0ORO1"	I 358.0	BOOL	// (A0RB.E5): ORDRE OUTIL 1
"A0ORO2"	I 358.1	BOOL	// (A0RB.E5): ORDRE OUTIL 2
"A0ORO3"	I 358.2	BOOL	// (A0RB.E5): ORDRE OUTIL 3
"A0ORO4"	I 358.3	BOOL	// (A0RB.E5): ORDRE OUTIL 4
"A0ORO5"	I 358.4	BOOL	// (A0RB.E5): ORDRE OUTIL 5
"A0ORO6"	I 358.5	BOOL	// (A0RB.E5): ORDRE OUTIL 6
"A0ORO7"	I 358.6	BOOL	// (A0RB.E5): ORDRE OUTIL 7
"A0ORO8"	I 358.7	BOOL	// (A0RB.E5): ORDRE OUTIL 8
"A0ORO9"	I 359.0	BOOL	// (A0RB.E5): ORDRE OUTIL 9
"A0ORO10"	I 359.1	BOOL	// (A0RB.E5): ORDRE OUTIL 10
"A0ORO11"	I 359.2	BOOL	// (A0RB.E5): ORDRE OUTIL 11
"A0ORO12"	I 359.3	BOOL	// (A0RB.E5): ORDRE OUTIL 12
"A0ORO13"	I 359.4	BOOL	// (A0RB.E5): ORDRE OUTIL 13
"A0ORO14"	I 359.5	BOOL	// (A0RB.E5): ORDRE OUTIL 14
"A0ORO15"	I 359.6	BOOL	// (A0RB.E5): ORDRE OUTIL 15
"A0ORO16"	I 359.7	BOOL	// (A0RB.E5): ORDRE OUTIL 16
"A0OR17"	I 364.0	BOOL	// (A0RB.E8): ORDRE 17
"A0OR18"	I 364.1	BOOL	// (A0RB.E8): ORDRE 18
"A0OR19"	I 364.2	BOOL	// (A0RB.E8): ORDRE 19
"A0OR20"	I 364.3	BOOL	// (A0RB.E8): ORDRE 20
"A0OR21"	I 364.4	BOOL	// (A0RB.E8): ORDRE 21
"A0OR22"	I 364.5	BOOL	// (A0RB.E8): ORDRE 22
"A0OR23"	I 364.6	BOOL	// (A0RB.E8): ORDRE 23
"A0OR24"	I 364.7	BOOL	// (A0RB.E8): ORDRE 24
"A0OR25"	I 365.0	BOOL	// (A0RB.E8): ORDRE 25
"A0OR26"	I 365.1	BOOL	// (A0RB.E8): ORDRE 26
"A0OR27"	I 365.2	BOOL	// (A0RB.E8): ORDRE 27
"A0OR28"	I 365.3	BOOL	// (A0RB.E8): ORDRE 28
"A0OR29"	I 365.4	BOOL	// (A0RB.E8): ORDRE 29
"A0OR30"	I 365.5	BOOL	// (A0RB.E8): ORDRE 30
"A0OR31"	I 365.6	BOOL	// (A0RB.E8): ORDRE 31
"A0OR32"	I 365.7	BOOL	// (A0RB.E8): ORDRE 32
"C0CDOB1"	I 430.0	BOOL	// (C0CIM.E1): DETECTEUR OUVERTURE BUTEE 1
"C0CDSPB1"	I 430.1	BOOL	// (C0CIM.E1): DETECTEUR SUPPORT PRESENT BUTEE 1
"C0CDOB2"	I 430.2	BOOL	// (C0CIM.E1): DETECTEUR OUVERTURE BUTEE 2
"C0CDSPB2"	I 430.3	BOOL	// (C0CIM.E1): DETECTEUR SUPPORT PRESENT BUTEE 2
"C0CDFB1"	I 430.4	BOOL	// (C0CIM.E1): DETECTEUR FERMETURE BUTEE 1
"C0CDSMAX"	I 430.5	BOOL	// (C0CIM.E1): DETECTEUR SEUIL MAX
"C0CDFB2"	I 430.6	BOOL	// (C0CIM.E1): DETECTEUR FERMETURE BUTEE 2
"C0CDDZB2"	I 430.7	BOOL	// (C0CIM.E1): DETECTEUR DEVERROUILLAGE DE ZONE BUTEE 2
"C0DPP1B2"	I 431.0	BOOL	// (C0CIM.E2): DETECTEUR PRESENCE PIECE TYPE 1
"C0CSSC"	I 431.2	BOOL	// (C0CIM.E2): C0C SELECTEUR DE SECURITE
"C0DPP2B2"	I 431.4	BOOL	// (C0CIM.E2): DETECTEUR PRESENCE PIECE TYPE 2
"H0DSSD"	I 450.0	BOOL	// (H0DIM.I1): SELECTEUR DE SECURITE
"H0DDM1_OK"	I 451.0	BOOL	// (H0DIM.DME1): DEPART MOTEUR PRET
"H0DDM1_CDM"	I 451.1	BOOL	// (H0DIM.DME1): DEPART MOTEUR EN MARCHE
"H0DDM1_DF"	I 451.2	BOOL	// (H0DIM.DME1): DEPART MOTEUR EN DEFAUT
"H0DDM1_AL"	I 451.3	BOOL	// (H0DIM.DME1): DEPART MOTEUR EN ALARME
"H0DDOB8"	I 453.0	BOOL	// (H0DIM.E1): DETECTEUR OUVERTURE BUTEE 8
"H0DDSPB8"	I 453.1	BOOL	// (H0DIM.E1): DETECTEUR SUPPORT PRESENT BUTEE 8
"H0DDOB9"	I 453.2	BOOL	// (H0DIM.E1): DETECTEUR OUVERTURE BUTEE 9
"H0DDSPB9"	I 453.3	BOOL	// (H0DIM.E1): DETECTEUR SUPPORT PRESENT BUTEE 9
"H0DDFB8"	I 453.4	BOOL	// (H0DIM.E1): DETECTEUR FERMETURE BUTEE 8
"H0DDSIL"	I 453.5	BOOL	// (H0DIM.E1): DETECTEUR SILHOUETTE
"H0DDFB9"	I 453.6	BOOL	// (H0DIM.E1): DETECTEUR FERMETURE BUTEE 9
"H0DDDZB9"	I 453.7	BOOL	// (H0DIM.E1): DETECTEUR DEVERROUILLAGE DE ZONE BUTEE 9
"H0DPP1B9"	I 454.0	BOOL	// (H0DIM.E2): DETECTEUR PRESENCE PIECE TYPE 1
"H0DDSMIN"	I 454.2	BOOL	// (H0DIM.E2): DETECTEUR SEUIL MIN
"H0DSSP"	I 454.3	BOOL	// (H0DIM.E2): SELECTEUR DE SECURITE
"H0DPP2B9"	I 454.4	BOOL	// (H0DIM.E2): DETECTEUR PRESENCE PIECE TYPE 2
"H0DDSMAX"	I 454.6	BOOL	// (H0DIM.E2): DETECTEUR SEUIL MAX
"H0DLIMEF"	I 454.7	BOOL	// (H0DIM.E2): LIMITEUR D'EFFORT
"Z1RB1CCB24Z"	I 470.4	BOOL	// (Z1RB1.M02): RETOUR CONTROLE DISJONCTEUR 24V (24Z)
"Z1RB1CCB24R"	I 470.5	BOOL	// (Z1RB1.M02): RETOUR CONTROLE DISJONCTEUR 24V (24R)
"A0BAU"	I 471.0	BOOL	// (Z1RB1.M05): ARRET D'URGENCE ROBOT
"A0RBMS1"	IW 350	WORD	// WORD 1 GENERAL DATA / GENERALITES
"A0RBMS2"	IW 352	WORD	// WORD 2 ROBOT ORDERS / ORDRES ROBOT
"A0RBMS3"	IW 354	WORD	// WORD 3 GRIPPER AND TOOL CHANGER / PREHENSEUR ET CHANGEUR OUTIL
"A0RBMS4"	IW 356	WORD	// WORD 4 FAULT NUMBER / NUMERO DE DEFAUT
"A0RBMS5"	IW 358	WORD	// WORD 5 TOOL ORDERS/ ORDRES OUTIL
"A0RBMS6"	IW 360	WORD	// WORD 6
"A0RBMS7"	IW 362	WORD	// WORD 7
"A0RBMS8"	IW 364	WORD	// WORD 8
"BA0"	M 0.0	BOOL	// FACILITY: BIT ALWAYS OFF / ILOT: BIT TOUJOURS A 0
"BA1"	M 0.1	BOOL	// FACILITY: BIT ALWAYS ON / ILOT: BIT TOUJOURS A 1
"BA1LIEN"	M 0.2	BOOL	// FACILITY: BIT ALWAYS ON (LINK IN THE PROGRAMMING NETWORK)
"SHUNT"	M 0.3	BOOL	// BIT FOR BYPASS DURING FACILITY START UP / BIT SHUNT POUR LA MISE AU POINT
"PERSO"	M 0.4	BOOL	// NEED TO PERSONALIZE BY THE PROGRAMMER / EQUATION A PERSONNALISER
"POUB"	M 0.5	BOOL	// DUST BIN BIT / BIT POUBELLE
"SYSFROID"	M 0.7	BOOL	// DETECTING COLD START PLC (OB102) / DETECTION DEMARRAGE A FROID API (OB102)
"ICL080S"	M 1.4	BOOL	// BLINKING INFORMATION / INFORMATION CLIGNOTEMENT
"IADF"	M 10.1	BOOL	// FACILITY: FAULT RESET INFORMATION (SAFETY)
"IR"	M 10.2	BOOL	// FACILITY: CONTROL ON INFORMATION (SAFETY)
"Z1DEF_MAJ"	M 11.0	BOOL	// ZONE 1: MAJOR FAULT (SAFETY)
"Z1IADF"	M 11.1	BOOL	// ZONE 1: FAULT RESET INFORMATION (SAFETY)
"Z1IR"	M 11.2	BOOL	// ZONE 1: CONTROL ON INFORMATION (SAFETY)
"Z1IAFJ"	M 11.3	BOOL	// ZONE 1: END OF PRODUCTION STOP INFORMATION (SAFETY)
"Z1MAUTO"	M 11.4	BOOL	// ZONE 1: ZONE IN AUTOMATIC MODE (SAFETY)
"H0AV"	M 100.0	BOOL	// Pilotage chaine H0
"SIMU"	M 105.0	BOOL	// Mode simulation en cours
"CYCL_EXC"	OB 1	OB 1	// EXECUTION CYCLE
"CYC_INT4"	OB 34	OB 34	// CYCLIC INTERRUPT 4
"I/O_FLT1"	OB 82	OB 82	// I/O POINT FAULT 1
"I/O_FLT2"	OB 83	OB 83	// I/O POINT FAULT 2
"OBNL_FLT"	OB 85	OB 85	// OB NOT LOADED FAULT
"RACK_FLT"	OB 86	OB 86	// LOSS OF RACK FAULT
"COMPLETE RESTART"	OB 100	OB 100	// COMPLETE RESTART
"MOD_ERR"	OB 122	OB 122	// MODULE ACCESS ERROR
"VADI"	Q 0.0	BOOL	// (MOP-IM.M06-07): VOYANT ANNULATION DEFAUT
"VMCY"	Q 0.1	BOOL	// (MOP-IM.M06-07): VOYANT MARCHE CYCLE
"VAOP"	Q 0.3	BOOL	// (MOP-IM.M06-07): VERRINE APPEL OPERATEUR
"A01EFSR1"	Q 56.0	BOOL	// (A01IM.S1): EV FERMETURE SERRAGE 1
"A01EFSR2"	Q 56.1	BOOL	// (A01IM.S1): A01 EV FERMETURE SERRAGE 2
"A01EFSR3"	Q 56.2	BOOL	// (A01IM.S1): A01 EV FERMETURE SERRAGE 3
"A01EOSR1"	Q 56.4	BOOL	// (A01IM.S1): A01 OUVERTURE SERRAGE 1
"A01EOSR2"	Q 56.5	BOOL	// (A01IM.S1): A01 EV OUVERTURE SERRAGE 2
"A01EOSR3"	Q 56.6	BOOL	// (A01IM.S1): A01 EV OUVERTURE SERRAGE 3
"B0EAPL1"	Q 58.0	BOOL	// (B0IM.B0S1): B0 EV AVANCE PILOTE 1
"B0EAPL2"	Q 58.1	BOOL	// (B0IM.B0S1): B0 EV AVANCE PILOTE 2
"B0EFSR3"	Q 58.2	BOOL	// (B0IM.B0S1): B0 EV FERMETURE SERRAGE 3
"B0EFSR4"	Q 58.3	BOOL	// (B0IM.B0S1): B0 EV FERMETURE SERRAGE 4
"B0ERPL1"	Q 58.4	BOOL	// (B0IM.B0S1): B0 EV RECUL PILOTE 1
"B0ERPL2"	Q 58.5	BOOL	// (B0IM.B0S1): B0 EV RECUL PILOTE 2
"B0EOSR3"	Q 58.6	BOOL	// (B0IM.B0S1): B0 EV OUVERTURE SERRAGE 3
"B0EOSR4"	Q 58.7	BOOL	// (B0IM.B0S1): B0 EV OUVERTURE SERRAGE 4
"Z1VMCY"	Q 200.0	BOOL	// (Z1ZB.M05): VOYANT MARCHE CYCLE
"Z1RCM"	Q 200.7	BOOL	// (Z1ZB.M05): RELAIS DE CONTROLE DE MASSE
"Z1RSC1"	Q 215.0	BOOL	// (Z1ZB.M09): RELAI COMMUN DE SECURITE SC1
"Z1RES"	Q 215.1	BOOL	// (Z1ZB.M09): RELAI COMMUN DE SECURITE ES
"Z1RFZ"	Q 215.2	BOOL	// (Z1ZB.M09): RELAI COMMUN DE SECURITE FZ
"Z1SPA1VMCY"	Q 300.7	BOOL	// (Z1SPA1.O0): VOYANT MARCHE CYCLE
"Z1SPA1VDACY"	Q 301.0	BOOL	// (Z1SPA1.O1): VOYANT DEMANDE ARRET CYCLE
"A0AEVRB"	Q 350.0	BOOL	// (A0RB.S1): AUTORISATION D'EVOLUTION
"A0DMSP"	Q 350.1	BOOL	// (A0RB.S1): DEMANDE DE MISE SOUS PUISSANCE
"A0STOP"	Q 350.2	BOOL	// (A0RB.S1): ARRET ROBOT
"A0DDCY"	Q 350.3	BOOL	// (A0RB.S1): DEPART CYCLE
"A0DEV"	Q 350.4	BOOL	// (A0RB.S1): DEVERMINAGE
"A0CVC_0"	Q 350.5	BOOL	// (A0RB.S1): CONTROLE VALIDATION CODE A 0
"A0CVC_1"	Q 350.6	BOOL	// (A0RB.S1): CONTROLE VALIDATION CODE A 1
"A0CPCO"	Q 350.7	BOOL	// (A0RB.S1): CONTOLE PARITE CODE
"A0C1"	Q 351.0	BOOL	// (A0RB.S1): CODE POIDS 1
"A0C2"	Q 351.1	BOOL	// (A0RB.S1): CODE POIDS 2
"A0C4"	Q 351.2	BOOL	// (A0RB.S1): CODE POIDS 4
"A0C8"	Q 351.3	BOOL	// (A0RB.S1): CODE POIDS 8
"A0C16"	Q 351.4	BOOL	// (A0RB.S1): CODE POIDS 16
"A0C32"	Q 351.5	BOOL	// (A0RB.S1): CODE POIDS 32
"A0C64"	Q 351.6	BOOL	// (A0RB.S1): CODE POIDS 64
"A0C128"	Q 351.7	BOOL	// (A0RB.S1): CODE POIDS 128
"A0EV1"	Q 352.0	BOOL	// (A0RB.S2): EVENEMENT 1
"A0EV2"	Q 352.1	BOOL	// (A0RB.S2): EVENEMENT 2
"A0EV3"	Q 352.2	BOOL	// (A0RB.S2): EVENEMENT 3
"A0EV4"	Q 352.3	BOOL	// (A0RB.S2): EVENEMENT 4
"A0EV5"	Q 352.4	BOOL	// (A0RB.S2): EVENEMENT 5
"A0EV6"	Q 352.5	BOOL	// (A0RB.S2): EVENEMENT 6
"A0EV7"	Q 352.6	BOOL	// (A0RB.S2): EVENEMENT 7
"A0EV8"	Q 352.7	BOOL	// (A0RB.S2): EVENEMENT 8
"A0EV9"	Q 353.0	BOOL	// (A0RB.S2): EVENEMENT 9
"A0EV10"	Q 353.1	BOOL	// (A0RB.S2): EVENEMENT 10
"A0EV11"	Q 353.2	BOOL	// (A0RB.S2): EVENEMENT 11
"A0EV12"	Q 353.3	BOOL	// (A0RB.S2): EVENEMENT 12
"A0EV13"	Q 353.4	BOOL	// (A0RB.S2): EVENEMENT 13
"A0EV14"	Q 353.5	BOOL	// (A0RB.S2): EVENEMENT 14
"A0EV15"	Q 353.6	BOOL	// (A0RB.S2): EVENEMENT 15
"A0EV16"	Q 353.7	BOOL	// (A0RB.S2): EVENEMENT 16
"A0ENPRO"	Q 354.0	BOOL	// (A0RB.S3): EN PRODUCTION
"A0RFZ"	Q 354.1	BOOL	// (A0RB.S3): ZONE FERMEE
"A0GS1"	Q 356.0	BOOL	// (A0RB.S4): GROUPE SEQUENCE POIDS 1
"A0GS2"	Q 356.1	BOOL	// (A0RB.S4): GROUPE SEQUENCE POIDS 2
"A0GS4"	Q 356.2	BOOL	// (A0RB.S4): GROUPE SEQUENCE POIDS 4
"A0GS8"	Q 356.3	BOOL	// (A0RB.S4): GROUPE SEQUENCE POIDS 8
"A0E1_SRE"	Q 356.4	BOOL	// (A0RB.S4): INFO DETECTION RECUL SEQUENCE 1
"A0E1_SAV"	Q 356.5	BOOL	// (A0RB.S4): INFO DETECTION AVANCE SEQUENCE 1
"A0E2_SRE"	Q 356.6	BOOL	// (A0RB.S4): INFO DETECTION RECUL SEQUENCE 2
"A0E2_SAV"	Q 356.7	BOOL	// (A0RB.S4): INFO DETECTION AVANCE SEQUENCE 2
"A0DECH"	Q 357.0	BOOL	// (A0RB.S4): COMMANDE DEVERROUILLAGE CHANGEUR
"A0EVO1"	Q 358.0	BOOL	// (A0RB.S5): EVENEMENT OUTIL 1
"A0EVO2"	Q 358.1	BOOL	// (A0RB.S5): EVENEMENT OUTIL 2
"A0EVO3"	Q 358.2	BOOL	// (A0RB.S5): EVENEMENT OUTIL 3
"A0EVO4"	Q 358.3	BOOL	// (A0RB.S5): EVENEMENT OUTIL 4
"A0EVO5"	Q 358.4	BOOL	// (A0RB.S5): EVENEMENT OUTIL 5
"A0EVO6"	Q 358.5	BOOL	// (A0RB.S5): EVENEMENT OUTIL 6
"A0EVO7"	Q 358.6	BOOL	// (A0RB.S5): EVENEMENT OUTIL 7
"A0EVO8"	Q 358.7	BOOL	// (A0RB.S5): EVENEMENT OUTIL 8
"A0EVO9"	Q 359.0	BOOL	// (A0RB.S5): EVENEMENT OUTIL 9
"A0EVO10"	Q 359.1	BOOL	// (A0RB.S5): EVENEMENT OUTIL 10
"A0EVO11"	Q 359.2	BOOL	// (A0RB.S5): EVENEMENT OUTIL 11
"A0EVO12"	Q 359.3	BOOL	// (A0RB.S5): EVENEMENT OUTIL 12
"A0EVO13"	Q 359.4	BOOL	// (A0RB.S5): EVENEMENT OUTIL 13
"A0EVO14"	Q 359.5	BOOL	// (A0RB.S5): EVENEMENT OUTIL 14
"A0EVO15"	Q 359.6	BOOL	// (A0RB.S5): EVENEMENT OUTIL 15
"A0EVO16"	Q 359.7	BOOL	// (A0RB.S5): EVENEMENT OUTIL 16
"A0EV17"	Q 364.0	BOOL	// (A0RB.S8): EVENEMENT 17
"A0EV18"	Q 364.1	BOOL	// (A0RB.S8): EVENEMENT 18
"A0EV19"	Q 364.2	BOOL	// (A0RB.S8): EVENEMENT 19
"A0EV20"	Q 364.3	BOOL	// (A0RB.S8): EVENEMENT 20
"A0EV21"	Q 364.4	BOOL	// (A0RB.S8): EVENEMENT 21
"A0EV22"	Q 364.5	BOOL	// (A0RB.S8): EVENEMENT 22
"A0EV23"	Q 364.6	BOOL	// (A0RB.S8): EVENEMENT 23
"A0EV24"	Q 364.7	BOOL	// (A0RB.S8): EVENEMENT 24
"A0EV25"	Q 365.0	BOOL	// (A0RB.S8): EVENEMENT 25
"A0EV26"	Q 365.1	BOOL	// (A0RB.S8): EVENEMENT 26
"A0EV27"	Q 365.2	BOOL	// (A0RB.S8): EVENEMENT 27
"A0EV28"	Q 365.3	BOOL	// (A0RB.S8): EVENEMENT 28
"A0EV29"	Q 365.4	BOOL	// (A0RB.S8): EVENEMENT 29
"A0EV30"	Q 365.5	BOOL	// (A0RB.S8): EVENEMENT 30
"A0EV31"	Q 365.6	BOOL	// (A0RB.S8): EVENEMENT 31
"A0EV32"	Q 365.7	BOOL	// (A0RB.S8): EVENEMENT 32
"C0CEOB1"	Q 430.0	BOOL	// (C0CIM.S1): ELECTROVANNE OUVERTURE BUTEE 1
"C0CEOB2"	Q 430.1	BOOL	// (C0CIM.S1): ELECTROVANNE OUVERTURE BUTEE 2
"C0CEFB1"	Q 430.4	BOOL	// (C0CIM.S1): ELECTROVANNE FERMETURE BUTEE 1
"C0CEFB2"	Q 430.5	BOOL	// (C0CIM.S1): ELECTROVANNE FERMETURE BUTEE 2
"H0DDM1_OAV"	Q 451.0	BOOL	// (H0DIM.DMS1): RELAI MARCHE AVANCE DEPART MOTEUR
"H0DDM1_ORE"	Q 451.1	BOOL	// (H0DIM.DMS1): RELAI MARCHE RECUL DEPART MOTEUR
"H0DDM1_FRE"	Q 451.2	BOOL	// (H0DIM.DMS1): COMMANDE FREIN DEPART MOTEUR
"H0DDM1_IR"	Q 451.3	BOOL	// (H0DIM.DMS1): INFORMATION REARMEMENT DEPART MOTEUR
"H0DEOB8"	Q 453.0	BOOL	// (H0DIM.S1): ELECTROVANNE OUVERTURE BUTEE 8
"H0DEOB9"	Q 453.1	BOOL	// (H0DIM.S1): ELECTROVANNE OUVERTURE BUTEE 9
"H0DEFB8"	Q 453.4	BOOL	// (H0DIM.S1): ELECTROVANNE FERMETURE BUTEE 8
"H0DEFB9"	Q 453.5	BOOL	// (H0DIM.S1): ELECTROVANNE FERMETURE BUTEE 9
"A0RBME1"	QW 350	WORD	// WORD 1 GENERAL DATA AND CYCLE CODE / CODE CYCLE ET GENERALITES
"A0RBME2"	QW 352	WORD	// WORD 2 ROBOT EVENTS / EVENEMENTS ROBOT
"A0RBME3"	QW 354	WORD	// WORD 3 GENERAL DATAS / GENERALITES
"A0RBME4"	QW 356	WORD	// WORD 4 GRIPPER AND TOOL CHANGER / PREHENSEUR ET CHANGEUR OUTIL
"A0RBME5"	QW 358	WORD	// WORD 5 TOOL EVENTS / EVENEMENTS OUTIL
"A0RBME6"	QW 360	WORD	// WORD 6
"A0RBME7"	QW 362	WORD	// WORD 7
"A0RBME8"	QW 364	WORD	// WORD 8
"TP"	SFB 3	SFB 3	// GENERATE A PULSE
"TON"	SFB 4	SFB 4	// GENERATE AN ON DELAY
"TOF"	SFB 5	SFB 5	// GENERATE AN OFF DELAY
"RDREC"	SFB 52	SFB 52	// READ A PROCESS DATA RECORD
"WRREC"	SFB 53	SFB 53	// WRITE A PROCESS DATA RECORD
"RALRM"	SFB 54	SFB 54	// Receive Alarm Data
"SET_CLK"	SFC 0	SFC 0	// SET SYSTEM CLOCK
"READ_CLK"	SFC 1	SFC 1	// READ SYSTEM CLOCK
"RD_SINFO"	SFC 6	SFC 6	// READ OB START INFORMATION
"D_ACT_DP"	SFC 12	SFC 12	// DEACTIVATING AND ACTIVATING DP SLAVES
"DPRD_DAT"	SFC 14	SFC 14	// READ CONSISTENT DATA OF A STANDARD DP SLAVE
"DPWR_DAT"	SFC 15	SFC 15	// WRITE CONSISTENT DATA TO A STANDARD DP SLAVE
"ALARM_SQ"	SFC 17	SFC 17	// Generate Block-Related Messages with Acknowledgment
"BLKMOV"	SFC 20	SFC 20	// COPY VARIABLES
"FILL"	SFC 21	SFC 21	// INITIALIZE A MEMORY AREA
"TEST_DB"	SFC 24	SFC 24	// TEST DATA BLOCK
"DIS_AIRT"	SFC 41	SFC 41	// DELAY THE HIGHER PRIORITY INTERRUPTS AND ASYNCHRONOUS ERRORS
"EN_AIRT"	SFC 42	SFC 42	// ENABLE HIGHER PRIORITY INTERRUPTS AND ASYNCHRONOUS ERRORS
"STP"	SFC 46	SFC 46	// CHANGE THE CPU TO STOP
"RDSYSST"	SFC 51	SFC 51	// READ A SYSTEM STATUS LIST OR PARTIAL LIST
"WR_REC"	SFC 58	SFC 58	// WRITE DATA RECORD
"RD_REC"	SFC 59	SFC 59	// READ A DATA RECORD
"TIME_TCK"	SFC 64	SFC 64	// READ THE SYSTEM TIME
"GEO_LOG"	SFC 70	SFC 70	// DETERMINE LOGICAL ADDRESS
"READ_DBL"	SFC 83	SFC 83	// READ DATA BLOCK OUT OF LOAD MEMORY
"WRIT_DBL"	SFC 84	SFC 84	// WRITE DATA BLOCK IN LOAD MEMORY
"DEL_SI"	SFC 106	SFC 106	// Deleting Dynamically Assigned System Instances
"ALARM_DQ"	SFC 107	SFC 107	// Creating Acknowledgeable Block-related Message
"ALARM_D"	SFC 108	SFC 108	// Creating Acknowledged Block-related Message
"LIEN_PUP"	UDT 1988	UDT 1988	// Gestion des Modes et des pupitres de cde manu de la  zone (BF_ZONE_MODE_IHM)
"LIEN_ILOT"	UDT 2004	UDT 2004	// INFO CONTROL LINKED TO THE FACILITY (BF_ILOT)
"MOT_FONC_MP"	UDT 2041	UDT 2041	// INFO CONTROL OF A MOVEMENT (BF_MOUVMP1)
"MOT_FONC"	UDT 2042	UDT 2042	// INFO D'UN MOUVEMENT (BF_MOUV2P1,BF_MVSE2P1, BF_RB_COD_PREH_API)
"VAT_SIMU"	VAT 1	
"Essais"	VAT 2	
END_SYMBOL_TABLE
